LIN {X 0,Y 368.852,Z 294.537,A -85,B 0,C 180,E1 -12651.37,E2 -12651.37} C_VEL
LIN {X 0,Y 368.906,Z 294.528,A -85,B 0,C 180,E1 -12655.15,E2 -12655.15} C_VEL
LIN {X 0,Y 368.892,Z 294.531,A -85,B 0,C 180,E1 -12659.049,E2 -12659.049} C_VEL
LIN {X 0,Y 368.954,Z 294.672,A -85,B 0,C 180,E1 -12660.004,E2 -12660.004} C_VEL
LIN {X 0,Y 372.447,Z 310.54,A -85,B 0,C 180,E1 -12663.38,E2 -12663.38} C_VEL
LIN {X 0,Y 373.826,Z 317.106,A -85,B 0,C 180,E1 -12664.734,E2 -12664.734} C_VEL
LIN {X 0,Y 372.805,Z 329.127,A -85,B 0,C 180,E1 -12666.984,E2 -12666.984} C_VEL
LIN {X 0,Y 371.4,Z 344.319,A -85,B 0,C 180,E1 -12669.802,E2 -12669.802} C_VEL
LIN {X 0,Y 374.275,Z 369.679,A -85,B 0,C 180,E1 -12670.516,E2 -12670.516} C_VEL
LIN {X 0,Y 372.854,Z 448.591,A -85,B 0,C 180,E1 -12672.239,E2 -12672.239} C_VEL
LIN {X 0,Y 372.479,Z 458.52,A -85,B 0,C 180,E1 -12672.575,E2 -12672.575} C_VEL
LIN {X 0,Y 371.991,Z 468.474,A -85,B 0,C 180,E1 -12673.047,E2 -12673.047} C_VEL
LIN {X 0,Y 371.44,Z 478.285,A -85,B 0,C 180,E1 -12673.657,E2 -12673.657} C_VEL
LIN {X 0,Y 370.84,Z 487.072,A -85,B 0,C 180,E1 -12674.336,E2 -12674.336} C_VEL
LIN {X 0,Y 370.263,Z 496.307,A -85,B 0,C 180,E1 -12675.213,E2 -12675.213} C_VEL
LIN {X 0,Y 369.643,Z 505.373,A -85,B 0,C 180,E1 -12676.26,E2 -12676.26} C_VEL
LIN {X 0,Y 369.043,Z 513.274,A -85,B 0,C 180,E1 -12677.353,E2 -12677.353} C_VEL
LIN {X 0,Y 368.613,Z 520.037,A -85,B 0,C 180,E1 -12678.455,E2 -12678.455} C_VEL
LIN {X 0,Y 368.156,Z 527.063,A -85,B 0,C 180,E1 -12679.833,E2 -12679.833} C_VEL
LIN {X 0,Y 367.85,Z 532.892,A -85,B 0,C 180,E1 -12681.211,E2 -12681.211} C_VEL
LIN {X 0,Y 367.65,Z 538.484,A -85,B 0,C 180,E1 -12682.865,E2 -12682.865} C_VEL
LIN {X 0,Y 367.522,Z 542.81,A -85,B 0,C 180,E1 -12684.516,E2 -12684.516} C_VEL
LIN {X 0,Y 367.546,Z 545.139,A -85,B 0,C 180,E1 -12685.616,E2 -12685.616} C_VEL
LIN {X 0,Y 367.621,Z 548.134,A -85,B 0,C 180,E1 -12687.811,E2 -12687.811} C_VEL
LIN {X 0,Y 367.594,Z 549.066,A -85,B 0,C 180,E1 -12688.907,E2 -12688.907} C_VEL
LIN {X 0,Y 367.581,Z 549.404,A -85,B 0,C 180,E1 -12691.098,E2 -12691.098} C_VEL
LIN {X 0,Y 367.525,Z 549.003,A -85,B 0,C 180,E1 -12692.194,E2 -12692.194} C_VEL
LIN {X 0,Y 367.479,Z 546.759,A -85,B 0,C 180,E1 -12694.389,E2 -12694.389} C_VEL
LIN {X 0,Y 367.484,Z 543.958,A -85,B 0,C 180,E1 -12696.027,E2 -12696.027} C_VEL
LIN {X 0,Y 367.679,Z 540.021,A -85,B 0,C 180,E1 -12697.691,E2 -12697.691} C_VEL
LIN {X 0,Y 367.968,Z 534.919,A -85,B 0,C 180,E1 -12699.344,E2 -12699.344} C_VEL
LIN {X 0,Y 368.394,Z 529.681,A -85,B 0,C 180,E1 -12700.721,E2 -12700.721} C_VEL
LIN {X 0,Y 369.051,Z 523.384,A -85,B 0,C 180,E1 -12702.093,E2 -12702.093} C_VEL
LIN {X 0,Y 369.786,Z 515.786,A -85,B 0,C 180,E1 -12703.464,E2 -12703.464} C_VEL
LIN {X 0,Y 370.598,Z 507.776,A -85,B 0,C 180,E1 -12704.666,E2 -12704.666} C_VEL
LIN {X 0,Y 371.53,Z 498.815,A -85,B 0,C 180,E1 -12705.779,E2 -12705.779} C_VEL
LIN {X 0,Y 372.409,Z 489.59,A -85,B 0,C 180,E1 -12706.726,E2 -12706.726} C_VEL
LIN {X 0,Y 373.338,Z 479.941,A -85,B 0,C 180,E1 -12707.53,E2 -12707.53} C_VEL
LIN {X 0,Y 374.156,Z 469.906,A -85,B 0,C 180,E1 -12708.197,E2 -12708.197} C_VEL
LIN {X 0,Y 374.823,Z 459.494,A -85,B 0,C 180,E1 -12708.73,E2 -12708.73} C_VEL
LIN {X 0,Y 375.383,Z 449.742,A -85,B 0,C 180,E1 -12709.09,E2 -12709.09} C_VEL
LIN {X 0,Y 376.048,Z 423.849,A -85,B 0,C 180,E1 -12709.706,E2 -12709.706} C_VEL
LIN {X 0,Y 377.433,Z 369.357,A -85,B 0,C 180,E1 -12710.955,E2 -12710.955} C_VEL
LIN {X 0,Y 374.759,Z 350.204,A -85,B 0,C 180,E1 -12711.646,E2 -12711.646} C_VEL
LIN {X 0,Y 373.55,Z 343.29,A -85,B 0,C 180,E1 -12711.944,E2 -12711.944} C_VEL
LIN {X 0,Y 375.579,Z 321.567,A -85,B 0,C 180,E1 -12715.738,E2 -12715.738} C_VEL
LIN {X 0,Y 374.001,Z 312.86,A -85,B 0,C 180,E1 -12717.513,E2 -12717.513} C_VEL
LIN {X 0,Y 371.33,Z 302.495,A -85,B 0,C 180,E1 -12719.789,E2 -12719.789} C_VEL
LIN {X 0,Y 368.908,Z 294.535,A -85,B 0,C 180,E1 -12721.713,E2 -12721.713} C_VEL
LIN {X 0,Y 368.921,Z 294.532,A -85,B 0,C 180,E1 -12725.001,E2 -12725.001} C_VEL
LIN {X 0,Y 368.899,Z 294.537,A -85,B 0,C 180,E1 -12728.639,E2 -12728.639} C_VEL
LIN {X 0,Y 368.871,Z 294.539,A -85,B 0,C 180,E1 -12732.008,E2 -12732.008} C_VEL
LIN {X 0,Y 368.868,Z 294.539,A -85,B 0,C 180,E1 -12735.175,E2 -12735.175} C_VEL
LIN {X 0,Y 368.88,Z 294.535,A -85,B 0,C 180,E1 -12738.178,E2 -12738.178} C_VEL
LIN {X 0,Y 368.897,Z 294.533,A -85,B 0,C 180,E1 -12741.358,E2 -12741.358} C_VEL
LIN {X 0,Y 368.92,Z 294.523,A -85,B 0,C 180,E1 -12745.145,E2 -12745.145} C_VEL
LIN {X 0,Y 368.913,Z 294.522,A -85,B 0,C 180,E1 -12749.046,E2 -12749.046} C_VEL
LIN {X 0,Y 368.962,Z 294.518,A -85,B 0,C 180,E1 -12751.563,E2 -12751.563} C_VEL
LIN {X 0,Y 368.94,Z 294.527,A -85,B 0,C 180,E1 -12755.224,E2 -12755.224} C_VEL
LIN {X 0,Y 368.951,Z 294.526,A -85,B 0,C 180,E1 -12758.959,E2 -12758.959} C_VEL
LIN {X 0,Y 368.97,Z 294.525,A -85,B 0,C 180,E1 -12762.257,E2 -12762.257} C_VEL
LIN {X 0,Y 369.015,Z 294.518,A -85,B 0,C 180,E1 -12766.228,E2 -12766.228} C_VEL
LIN {X 0,Y 369.046,Z 294.519,A -85,B 0,C 180,E1 -12770.132,E2 -12770.132} C_VEL
LIN {X 0,Y 369.16,Z 294.554,A -85,B 0,C 180,E1 -12772.652,E2 -12772.652} C_VEL
LIN {X 0,Y 371.658,Z 303.249,A -85,B 0,C 180,E1 -12774.575,E2 -12774.575} C_VEL
LIN {X 0,Y 373.879,Z 311.472,A -85,B 0,C 180,E1 -12776.31,E2 -12776.31} C_VEL
LIN {X 0,Y 372.861,Z 329.538,A -85,B 0,C 180,E1 -12779.461,E2 -12779.461} C_VEL
LIN {X 0,Y 372.43,Z 338.244,A -85,B 0,C 180,E1 -12780.974,E2 -12780.974} C_VEL
LIN {X 0,Y 375.936,Z 356.545,A -85,B 0,C 180,E1 -12781.789,E2 -12781.789} C_VEL
LIN {X 0,Y 377.093,Z 364.499,A -85,B 0,C 180,E1 -12782.108,E2 -12782.108} C_VEL
LIN {X 0,Y 375.003,Z 424.893,A -85,B 0,C 180,E1 -12783.728,E2 -12783.728} C_VEL
LIN {X 0,Y 374.491,Z 435.675,A -85,B 0,C 180,E1 -12784.171,E2 -12784.171} C_VEL
LIN {X 0,Y 373.795,Z 447.132,A -85,B 0,C 180,E1 -12784.842,E2 -12784.842} C_VEL
LIN {X 0,Y 373.077,Z 457.501,A -85,B 0,C 180,E1 -12785.676,E2 -12785.676} C_VEL
LIN {X 0,Y 372.37,Z 465.772,A -85,B 0,C 180,E1 -12786.503,E2 -12786.503} C_VEL
LIN {X 0,Y 371.6,Z 473.736,A -85,B 0,C 180,E1 -12787.472,E2 -12787.472} C_VEL
LIN {X 0,Y 370.891,Z 480.383,A -85,B 0,C 180,E1 -12788.445,E2 -12788.445} C_VEL
LIN {X 0,Y 370.263,Z 486.344,A -85,B 0,C 180,E1 -12789.489,E2 -12789.489} C_VEL
LIN {X 0,Y 369.628,Z 492.019,A -85,B 0,C 180,E1 -12790.684,E2 -12790.684} C_VEL
LIN {X 0,Y 369.249,Z 495.434,A -85,B 0,C 180,E1 -12791.529,E2 -12791.529} C_VEL
LIN {X 0,Y 368.793,Z 499.293,A -85,B 0,C 180,E1 -12792.66,E2 -12792.66} C_VEL
LIN {X 0,Y 368.434,Z 502.508,A -85,B 0,C 180,E1 -12793.828,E2 -12793.828} C_VEL
LIN {X 0,Y 368.016,Z 505.852,A -85,B 0,C 180,E1 -12795.508,E2 -12795.508} C_VEL
LIN {X 0,Y 367.719,Z 507.88,A -85,B 0,C 180,E1 -12797.145,E2 -12797.145} C_VEL
LIN {X 0,Y 367.609,Z 508.44,A -85,B 0,C 180,E1 -12797.812,E2 -12797.812} C_VEL
LIN {X 0,Y 367.475,Z 508.798,A -85,B 0,C 180,E1 -12798.974,E2 -12798.974} C_VEL
LIN {X 0,Y 367.448,Z 508.486,A -85,B 0,C 180,E1 -12800.423,E2 -12800.423} C_VEL
LIN {X 0,Y 367.429,Z 507.838,A -85,B 0,C 180,E1 -12801.311,E2 -12801.311} C_VEL
LIN {X 0,Y 367.55,Z 506.489,A -85,B 0,C 180,E1 -12802.485,E2 -12802.485} C_VEL
LIN {X 0,Y 367.696,Z 504.51,A -85,B 0,C 180,E1 -12803.666,E2 -12803.666} C_VEL
LIN {X 0,Y 367.829,Z 501.801,A -85,B 0,C 180,E1 -12804.857,E2 -12804.857} C_VEL
LIN {X 0,Y 368.046,Z 497.943,A -85,B 0,C 180,E1 -12806.177,E2 -12806.177} C_VEL
LIN {X 0,Y 368.437,Z 491.446,A -85,B 0,C 180,E1 -12807.863,E2 -12807.863} C_VEL
LIN {X 0,Y 368.84,Z 485.092,A -85,B 0,C 180,E1 -12809.165,E2 -12809.165} C_VEL
LIN {X 0,Y 369.281,Z 478.413,A -85,B 0,C 180,E1 -12810.288,E2 -12810.288} C_VEL
LIN {X 0,Y 369.782,Z 470.965,A -85,B 0,C 180,E1 -12811.326,E2 -12811.326} C_VEL
LIN {X 0,Y 370.357,Z 461.379,A -85,B 0,C 180,E1 -12812.418,E2 -12812.418} C_VEL
LIN {X 0,Y 370.87,Z 450.933,A -85,B 0,C 180,E1 -12813.337,E2 -12813.337} C_VEL
LIN {X 0,Y 371.343,Z 442.01,A -85,B 0,C 180,E1 -12813.95,E2 -12813.95} C_VEL
LIN {X 0,Y 371.712,Z 431.539,A -85,B 0,C 180,E1 -12814.496,E2 -12814.496} C_VEL
LIN {X 0,Y 371.961,Z 421.603,A -85,B 0,C 180,E1 -12814.86,E2 -12814.86} C_VEL
LIN {X 0,Y 373.105,Z 361.779,A -85,B 0,C 180,E1 -12816.312,E2 -12816.312} C_VEL
LIN {X 0,Y 370.041,Z 339.575,A -85,B 0,C 180,E1 -12816.982,E2 -12816.982} C_VEL
LIN {X 0,Y 370.885,Z 325.677,A -85,B 0,C 180,E1 -12820.112,E2 -12820.112} C_VEL
LIN {X 0,Y 371.83,Z 312.012,A -85,B 0,C 180,E1 -12823.249,E2 -12823.249} C_VEL
LIN {X 0,Y 371.695,Z 308.56,A -85,B 0,C 180,E1 -12824.072,E2 -12824.072} C_VEL
LIN {X 0,Y 369.089,Z 295.334,A -85,B 0,C 180,E1 -12827.423,E2 -12827.423} C_VEL
LIN {X 0,Y 368.917,Z 294.532,A -85,B 0,C 180,E1 -12827.657,E2 -12827.657} C_VEL
LIN {X 0,Y 368.873,Z 294.538,A -85,B 0,C 180,E1 -12831.368,E2 -12831.368} C_VEL
LIN {X 0,Y 368.928,Z 294.526,A -85,B 0,C 180,E1 -12835.147,E2 -12835.147} C_VEL
LIN {X 0,Y 368.896,Z 294.529,A -85,B 0,C 180,E1 -12839.044,E2 -12839.044} C_VEL
LIN {X 0,Y 368.908,Z 294.529,A -85,B 0,C 180,E1 -12841.558,E2 -12841.558} C_VEL
LIN {X 0,Y 368.921,Z 294.531,A -85,B 0,C 180,E1 -12844.014,E2 -12844.014} C_VEL
LIN {X 0,Y 368.899,Z 294.529,A -85,B 0,C 180,E1 -12847.603,E2 -12847.603} C_VEL
LIN {X 0,Y 368.953,Z 294.524,A -85,B 0,C 180,E1 -12851.105,E2 -12851.105} C_VEL
LIN {X 0,Y 368.998,Z 294.52,A -85,B 0,C 180,E1 -12854.535,E2 -12854.535} C_VEL
LIN {X 0,Y 369.063,Z 294.513,A -85,B 0,C 180,E1 -12856.79,E2 -12856.79} C_VEL
LIN {X 0,Y 369.065,Z 294.508,A -85,B 0,C 180,E1 -12860.13,E2 -12860.13} C_VEL
LIN {X 0,Y 369.16,Z 294.503,A -85,B 0,C 180,E1 -12863.439,E2 -12863.439} C_VEL
LIN {X 0,Y 369.299,Z 294.484,A -85,B 0,C 180,E1 -12867.817,E2 -12867.817} C_VEL
LIN {X 0,Y 369.205,Z 294.491,A -85,B 0,C 180,E1 -12871.088,E2 -12871.088} C_VEL
LIN {X 0,Y 369.298,Z 294.482,A -85,B 0,C 180,E1 -12872.179,E2 -12872.179} C_VEL
LIN {X 0,Y 369.156,Z 294.499,A -85,B 0,C 180,E1 -12876.556,E2 -12876.556} C_VEL
LIN {X 0,Y 369.06,Z 294.511,A -85,B 0,C 180,E1 -12879.865,E2 -12879.865} C_VEL
LIN {X 0,Y 369.036,Z 294.512,A -85,B 0,C 180,E1 -12883.769,E2 -12883.769} C_VEL
LIN {X 0,Y 368.962,Z 294.526,A -85,B 0,C 180,E1 -12886.694,E2 -12886.694} C_VEL
LIN {X 0,Y 368.276,Z 294.607,A -85,B 0,C 180,E1 -12887.604,E2 -12887.604} C_VEL
LIN {X 0,Y 365.402,Z 294.969,A -85,B 0,C 180,E1 -12889.084,E2 -12889.084} C_VEL
LIN {X 0,Y 362.976,Z 295.272,A -85,B 0,C 180,E1 -12890.281,E2 -12890.281} C_VEL
LIN {X 0,Y 361.934,Z 295.401,A -85,B 0,C 180,E1 -12891.207,E2 -12891.207} C_VEL
LIN {X 0,Y 361.849,Z 295.408,A -85,B 0,C 180,E1 -12891.521,E2 -12891.521} C_VEL
LIN {X 0,Y 361.873,Z 295.41,A -85,B 0,C 180,E1 -12895.289,E2 -12895.289} C_VEL
LIN {X 0,Y 361.843,Z 295.411,A -85,B 0,C 180,E1 -12899.069,E2 -12899.069} C_VEL
LIN {X 0,Y 361.833,Z 295.41,A -85,B 0,C 180,E1 -12902.94,E2 -12902.94} C_VEL
LIN {X 0,Y 361.85,Z 295.412,A -85,B 0,C 180,E1 -12905.632,E2 -12905.632} C_VEL
LIN {X 0,Y 361.843,Z 295.408,A -85,B 0,C 180,E1 -12909.02,E2 -12909.02} C_VEL
LIN {X 0,Y 361.809,Z 295.413,A -85,B 0,C 180,E1 -12912.824,E2 -12912.824} C_VEL
LIN {X 0,Y 361.79,Z 295.417,A -85,B 0,C 180,E1 -12915.942,E2 -12915.942} C_VEL
LIN {X 0,Y 361.804,Z 295.413,A -85,B 0,C 180,E1 -12919.24,E2 -12919.24} C_VEL
LIN {X 0,Y 361.827,Z 295.417,A -85,B 0,C 180,E1 -12922.773,E2 -12922.773} C_VEL
LIN {X 0,Y 361.814,Z 295.412,A -85,B 0,C 180,E1 -12925.715,E2 -12925.715} C_VEL
LIN {X 0,Y 361.837,Z 295.41,A -85,B 0,C 180,E1 -12929.668,E2 -12929.668} C_VEL
LIN {X 0,Y 361.913,Z 295.405,A -85,B 0,C 180,E1 -12933.471,E2 -12933.471} C_VEL
LIN {X 0,Y 361.834,Z 295.411,A -85,B 0,C 180,E1 -12937.14,E2 -12937.14} C_VEL
LIN {X 0,Y 361.82,Z 295.41,A -85,B 0,C 180,E1 -12940.718,E2 -12940.718} C_VEL
LIN {X 0,Y 361.895,Z 295.406,A -85,B 0,C 180,E1 -12944.223,E2 -12944.223} C_VEL
LIN {X 0,Y 361.951,Z 295.397,A -85,B 0,C 180,E1 -12946.525,E2 -12946.525} C_VEL
LIN {X 0,Y 361.984,Z 295.393,A -85,B 0,C 180,E1 -12949.936,E2 -12949.936} C_VEL
LIN {X 0,Y 362.112,Z 295.374,A -85,B 0,C 180,E1 -12953.312,E2 -12953.312} C_VEL
LIN {X 0,Y 362.236,Z 295.359,A -85,B 0,C 180,E1 -12957.776,E2 -12957.776} C_VEL
LIN {X 0,Y 362.374,Z 295.342,A -85,B 0,C 180,E1 -12959.999,E2 -12959.999} C_VEL
LIN {X 0,Y 362.23,Z 295.36,A -85,B 0,C 180,E1 -12962.223,E2 -12962.223} C_VEL
LIN {X 0,Y 362.111,Z 295.376,A -85,B 0,C 180,E1 -12966.687,E2 -12966.687} C_VEL
LIN {X 0,Y 361.981,Z 295.392,A -85,B 0,C 180,E1 -12970.063,E2 -12970.063} C_VEL
LIN {X 0,Y 361.949,Z 295.399,A -85,B 0,C 180,E1 -12973.899,E2 -12973.899} C_VEL
LIN {X 0,Y 361.92,Z 295.405,A -85,B 0,C 180,E1 -12977.94,E2 -12977.94} C_VEL
LIN {X 0,Y 361.837,Z 295.41,A -85,B 0,C 180,E1 -12981.656,E2 -12981.656} C_VEL
LIN {X 0,Y 361.882,Z 295.403,A -85,B 0,C 180,E1 -12985.293,E2 -12985.293} C_VEL
LIN {X 0,Y 361.862,Z 295.406,A -85,B 0,C 180,E1 -12987.782,E2 -12987.782} C_VEL
LIN {X 0,Y 361.792,Z 295.414,A -85,B 0,C 180,E1 -12991.633,E2 -12991.633} C_VEL
LIN {X 0,Y 361.835,Z 295.411,A -85,B 0,C 180,E1 -12995.348,E2 -12995.348} C_VEL
LIN {X 0,Y 361.827,Z 295.416,A -85,B 0,C 180,E1 -12999.029,E2 -12999.029} C_VEL
LIN {X 0,Y 361.802,Z 295.415,A -85,B 0,C 180,E1 -13002.833,E2 -13002.833} C_VEL
LIN {X 0,Y 361.785,Z 295.417,A -85,B 0,C 180,E1 -13005.951,E2 -13005.951} C_VEL
LIN {X 0,Y 361.805,Z 295.415,A -85,B 0,C 180,E1 -13009.249,E2 -13009.249} C_VEL
LIN {X 0,Y 361.835,Z 295.409,A -85,B 0,C 180,E1 -13012.985,E2 -13012.985} C_VEL
LIN {X 0,Y 361.835,Z 295.411,A -85,B 0,C 180,E1 -13016.635,E2 -13016.635} C_VEL
LIN {X 0,Y 361.89,Z 295.489,A -85,B 0,C 180,E1 -13019.679,E2 -13019.679} C_VEL
LIN {X 0,Y 365.13,Z 310.229,A -85,B 0,C 180,E1 -13022.886,E2 -13022.886} C_VEL
LIN {X 0,Y 366.901,Z 318.921,A -85,B 0,C 180,E1 -13024.712,E2 -13024.712} C_VEL
LIN {X 0,Y 365.132,Z 337.578,A -85,B 0,C 180,E1 -13028.257,E2 -13028.257} C_VEL
LIN {X 0,Y 364.455,Z 344.417,A -85,B 0,C 180,E1 -13029.547,E2 -13029.547} C_VEL
LIN {X 0,Y 367.345,Z 370.807,A -85,B 0,C 180,E1 -13030.286,E2 -13030.286} C_VEL
LIN {X 0,Y 365.895,Z 448.793,A -85,B 0,C 180,E1 -13032.034,E2 -13032.034} C_VEL
LIN {X 0,Y 365.517,Z 458.547,A -85,B 0,C 180,E1 -13032.376,E2 -13032.376} C_VEL
LIN {X 0,Y 365.015,Z 468.409,A -85,B 0,C 180,E1 -13032.857,E2 -13032.857} C_VEL
LIN {X 0,Y 364.448,Z 478.164,A -85,B 0,C 180,E1 -13033.479,E2 -13033.479} C_VEL
LIN {X 0,Y 363.837,Z 486.913,A -85,B 0,C 180,E1 -13034.17,E2 -13034.17} C_VEL
LIN {X 0,Y 363.201,Z 496.869,A -85,B 0,C 180,E1 -13035.148,E2 -13035.148} C_VEL
LIN {X 0,Y 362.628,Z 504.665,A -85,B 0,C 180,E1 -13036.064,E2 -13036.064} C_VEL
LIN {X 0,Y 362.044,Z 512.174,A -85,B 0,C 180,E1 -13037.104,E2 -13037.104} C_VEL
LIN {X 0,Y 361.48,Z 520.509,A -85,B 0,C 180,E1 -13038.508,E2 -13038.508} C_VEL
LIN {X 0,Y 361.043,Z 527.396,A -85,B 0,C 180,E1 -13039.913,E2 -13039.913} C_VEL
LIN {X 0,Y 360.783,Z 532.112,A -85,B 0,C 180,E1 -13041.038,E2 -13041.038} C_VEL
LIN {X 0,Y 360.577,Z 537.794,A -85,B 0,C 180,E1 -13042.725,E2 -13042.725} C_VEL
LIN {X 0,Y 360.438,Z 542.193,A -85,B 0,C 180,E1 -13044.408,E2 -13044.408} C_VEL
LIN {X 0,Y 360.48,Z 544.54,A -85,B 0,C 180,E1 -13045.53,E2 -13045.53} C_VEL
LIN {X 0,Y 360.537,Z 547.644,A -85,B 0,C 180,E1 -13047.768,E2 -13047.768} C_VEL
LIN {X 0,Y 360.529,Z 548.586,A -85,B 0,C 180,E1 -13048.885,E2 -13048.885} C_VEL
LIN {X 0,Y 360.515,Z 549.019,A -85,B 0,C 180,E1 -13051.119,E2 -13051.119} C_VEL
LIN {X 0,Y 360.427,Z 548.613,A -85,B 0,C 180,E1 -13052.237,E2 -13052.237} C_VEL
LIN {X 0,Y 360.386,Z 546.46,A -85,B 0,C 180,E1 -13054.476,E2 -13054.476} C_VEL
LIN {X 0,Y 360.382,Z 544.064,A -85,B 0,C 180,E1 -13055.975,E2 -13055.975} C_VEL
LIN {X 0,Y 360.607,Z 539.811,A -85,B 0,C 180,E1 -13057.843,E2 -13057.843} C_VEL
LIN {X 0,Y 360.931,Z 534.778,A -85,B 0,C 180,E1 -13059.528,E2 -13059.528} C_VEL
LIN {X 0,Y 361.388,Z 529.619,A -85,B 0,C 180,E1 -13060.931,E2 -13060.931} C_VEL
LIN {X 0,Y 362.098,Z 523.387,A -85,B 0,C 180,E1 -13062.329,E2 -13062.329} C_VEL
LIN {X 0,Y 362.863,Z 515.856,A -85,B 0,C 180,E1 -13063.726,E2 -13063.726} C_VEL
LIN {X 0,Y 363.711,Z 507.909,A -85,B 0,C 180,E1 -13064.952,E2 -13064.952} C_VEL
LIN {X 0,Y 364.717,Z 499.054,A -85,B 0,C 180,E1 -13066.082,E2 -13066.082} C_VEL
LIN {X 0,Y 365.651,Z 489.947,A -85,B 0,C 180,E1 -13067.045,E2 -13067.045} C_VEL
LIN {X 0,Y 366.618,Z 480.522,A -85,B 0,C 180,E1 -13067.862,E2 -13067.862} C_VEL
LIN {X 0,Y 367.561,Z 469.647,A -85,B 0,C 180,E1 -13068.607,E2 -13068.607} C_VEL
LIN {X 0,Y 368.26,Z 459.364,A -85,B 0,C 180,E1 -13069.148,E2 -13069.148} C_VEL
LIN {X 0,Y 368.867,Z 448.662,A -85,B 0,C 180,E1 -13069.55,E2 -13069.55} C_VEL
LIN {X 0,Y 369.763,Z 418.32,A -85,B 0,C 180,E1 -13070.272,E2 -13070.272} C_VEL
LIN {X 0,Y 371.004,Z 369.957,A -85,B 0,C 180,E1 -13071.415,E2 -13071.415} C_VEL
LIN {X 0,Y 368.495,Z 351.79,A -85,B 0,C 180,E1 -13072.101,E2 -13072.101} C_VEL
LIN {X 0,Y 366.974,Z 343.172,A -85,B 0,C 180,E1 -13072.489,E2 -13072.489} C_VEL
LIN {X 0,Y 368.932,Z 323.532,A -85,B 0,C 180,E1 -13075.985,E2 -13075.985} C_VEL
LIN {X 0,Y 367.259,Z 314.592,A -85,B 0,C 180,E1 -13077.873,E2 -13077.873} C_VEL
LIN {X 0,Y 364.349,Z 303.535,A -85,B 0,C 180,E1 -13080.405,E2 -13080.405} C_VEL
LIN {X 0,Y 361.852,Z 295.413,A -85,B 0,C 180,E1 -13082.447,E2 -13082.447} C_VEL
LIN {X 0,Y 361.86,Z 295.413,A -85,B 0,C 180,E1 -13085.636,E2 -13085.636} C_VEL
LIN {X 0,Y 361.86,Z 295.415,A -85,B 0,C 180,E1 -13089.026,E2 -13089.026} C_VEL
LIN {X 0,Y 361.826,Z 295.417,A -85,B 0,C 180,E1 -13092.828,E2 -13092.828} C_VEL
LIN {X 0,Y 361.806,Z 295.416,A -85,B 0,C 180,E1 -13095.946,E2 -13095.946} C_VEL
LIN {X 0,Y 361.856,Z 295.411,A -85,B 0,C 180,E1 -13099.238,E2 -13099.238} C_VEL
LIN {X 0,Y 361.853,Z 295.406,A -85,B 0,C 180,E1 -13102.981,E2 -13102.981} C_VEL
LIN {X 0,Y 361.842,Z 295.403,A -85,B 0,C 180,E1 -13106.63,E2 -13106.63} C_VEL
LIN {X 0,Y 361.858,Z 295.4,A -85,B 0,C 180,E1 -13109.671,E2 -13109.671} C_VEL
LIN {X 0,Y 361.935,Z 295.397,A -85,B 0,C 180,E1 -13113.474,E2 -13113.474} C_VEL
LIN {X 0,Y 361.888,Z 295.408,A -85,B 0,C 180,E1 -13117.145,E2 -13117.145} C_VEL
LIN {X 0,Y 361.911,Z 295.403,A -85,B 0,C 180,E1 -13120.724,E2 -13120.724} C_VEL
LIN {X 0,Y 361.923,Z 295.402,A -85,B 0,C 180,E1 -13124.226,E2 -13124.226} C_VEL
LIN {X 0,Y 361.977,Z 295.396,A -85,B 0,C 180,E1 -13126.528,E2 -13126.528} C_VEL
LIN {X 0,Y 362.01,Z 295.396,A -85,B 0,C 180,E1 -13129.938,E2 -13129.938} C_VEL
LIN {X 0,Y 362.135,Z 295.534,A -85,B 0,C 180,E1 -13131.954,E2 -13131.954} C_VEL
LIN {X 0,Y 365.035,Z 305.197,A -85,B 0,C 180,E1 -13134.199,E2 -13134.199} C_VEL
LIN {X 0,Y 367.348,Z 314.468,A -85,B 0,C 180,E1 -13136.2,E2 -13136.2} C_VEL
LIN {X 0,Y 366.089,Z 334.351,A -85,B 0,C 180,E1 -13139.726,E2 -13139.726} C_VEL
LIN {X 0,Y 365.832,Z 338.257,A -85,B 0,C 180,E1 -13140.413,E2 -13140.413} C_VEL
LIN {X 0,Y 369.455,Z 356.953,A -85,B 0,C 180,E1 -13141.304,E2 -13141.304} C_VEL
LIN {X 0,Y 370.657,Z 365.769,A -85,B 0,C 180,E1 -13141.663,E2 -13141.663} C_VEL
LIN {X 0,Y 368.478,Z 425.757,A -85,B 0,C 180,E1 -13143.315,E2 -13143.315} C_VEL
LIN {X 0,Y 367.891,Z 437.742,A -85,B 0,C 180,E1 -13143.834,E2 -13143.834} C_VEL
LIN {X 0,Y 367.057,Z 449.679,A -85,B 0,C 180,E1 -13144.608,E2 -13144.608} C_VEL
LIN {X 0,Y 366.383,Z 458.543,A -85,B 0,C 180,E1 -13145.356,E2 -13145.356} C_VEL
LIN {X 0,Y 365.615,Z 466.762,A -85,B 0,C 180,E1 -13146.208,E2 -13146.208} C_VEL
LIN {X 0,Y 364.783,Z 474.609,A -85,B 0,C 180,E1 -13147.195,E2 -13147.195} C_VEL
LIN {X 0,Y 363.949,Z 482.061,A -85,B 0,C 180,E1 -13148.328,E2 -13148.328} C_VEL
LIN {X 0,Y 363.068,Z 489.887,A -85,B 0,C 180,E1 -13149.805,E2 -13149.805} C_VEL
LIN {X 0,Y 362.375,Z 495.583,A -85,B 0,C 180,E1 -13151.184,E2 -13151.184} C_VEL
LIN {X 0,Y 361.858,Z 499.502,A -85,B 0,C 180,E1 -13152.336,E2 -13152.336} C_VEL
LIN {X 0,Y 361.343,Z 503.801,A -85,B 0,C 180,E1 -13154.014,E2 -13154.014} C_VEL
LIN {X 0,Y 360.868,Z 506.998,A -85,B 0,C 180,E1 -13155.823,E2 -13155.823} C_VEL
LIN {X 0,Y 360.613,Z 508.531,A -85,B 0,C 180,E1 -13157.272,E2 -13157.272} C_VEL
LIN {X 0,Y 360.475,Z 509.069,A -85,B 0,C 180,E1 -13158.177,E2 -13158.177} C_VEL
LIN {X 0,Y 360.377,Z 509.271,A -85,B 0,C 180,E1 -13159.362,E2 -13159.362} C_VEL
LIN {X 0,Y 360.357,Z 508.799,A -85,B 0,C 180,E1 -13160.596,E2 -13160.596} C_VEL
LIN {X 0,Y 360.388,Z 507.747,A -85,B 0,C 180,E1 -13161.748,E2 -13161.748} C_VEL
LIN {X 0,Y 360.598,Z 504.893,A -85,B 0,C 180,E1 -13163.656,E2 -13163.656} C_VEL
LIN {X 0,Y 360.806,Z 500.774,A -85,B 0,C 180,E1 -13165.375,E2 -13165.375} C_VEL
LIN {X 0,Y 361.123,Z 495.855,A -85,B 0,C 180,E1 -13166.904,E2 -13166.904} C_VEL
LIN {X 0,Y 361.414,Z 490.886,A -85,B 0,C 180,E1 -13168.136,E2 -13168.136} C_VEL
LIN {X 0,Y 361.814,Z 484.819,A -85,B 0,C 180,E1 -13169.372,E2 -13169.372} C_VEL
LIN {X 0,Y 362.406,Z 476.428,A -85,B 0,C 180,E1 -13170.763,E2 -13170.763} C_VEL
LIN {X 0,Y 363.011,Z 466.833,A -85,B 0,C 180,E1 -13172.005,E2 -13172.005} C_VEL
LIN {X 0,Y 363.587,Z 457.853,A -85,B 0,C 180,E1 -13172.933,E2 -13172.933} C_VEL
LIN {X 0,Y 364.052,Z 448.472,A -85,B 0,C 180,E1 -13173.713,E2 -13173.713} C_VEL
LIN {X 0,Y 364.484,Z 438.919,A -85,B 0,C 180,E1 -13174.334,E2 -13174.334} C_VEL
LIN {X 0,Y 364.902,Z 426.577,A -85,B 0,C 180,E1 -13174.917,E2 -13174.917} C_VEL
LIN {X 0,Y 365.329,Z 408.302,A -85,B 0,C 180,E1 -13175.413,E2 -13175.413} C_VEL
LIN {X 0,Y 366.145,Z 362.498,A -85,B 0,C 180,E1 -13176.544,E2 -13176.544} C_VEL
LIN {X 0,Y 363.116,Z 339.521,A -85,B 0,C 180,E1 -13177.274,E2 -13177.274} C_VEL
LIN {X 0,Y 364.293,Z 321.474,A -85,B 0,C 180,E1 -13181.422,E2 -13181.422} C_VEL
LIN {X 0,Y 364.866,Z 310.928,A -85,B 0,C 180,E1 -13183.903,E2 -13183.903} C_VEL
LIN {X 0,Y 362.627,Z 299.172,A -85,B 0,C 180,E1 -13186.91,E2 -13186.91} C_VEL
LIN {X 0,Y 361.855,Z 295.41,A -85,B 0,C 180,E1 -13187.916,E2 -13187.916} C_VEL
LIN {X 0,Y 361.839,Z 295.415,A -85,B 0,C 180,E1 -13191.573,E2 -13191.573} C_VEL
LIN {X 0,Y 361.868,Z 295.405,A -85,B 0,C 180,E1 -13194.658,E2 -13194.658} C_VEL
LIN {X 0,Y 361.834,Z 295.411,A -85,B 0,C 180,E1 -13198.371,E2 -13198.371} C_VEL
LIN {X 0,Y 361.85,Z 295.407,A -85,B 0,C 180,E1 -13200.951,E2 -13200.951} C_VEL
LIN {X 0,Y 361.854,Z 295.409,A -85,B 0,C 180,E1 -13204.705,E2 -13204.705} C_VEL
LIN {X 0,Y 361.857,Z 295.412,A -85,B 0,C 180,E1 -13208.345,E2 -13208.345} C_VEL
LIN {X 0,Y 361.924,Z 295.399,A -85,B 0,C 180,E1 -13212.085,E2 -13212.085} C_VEL
LIN {X 0,Y 362.004,Z 295.388,A -85,B 0,C 180,E1 -13216.101,E2 -13216.101} C_VEL
LIN {X 0,Y 362.002,Z 295.388,A -85,B 0,C 180,E1 -13219.936,E2 -13219.936} C_VEL
LIN {X 0,Y 362.124,Z 295.38,A -85,B 0,C 180,E1 -13223.311,E2 -13223.311} C_VEL
LIN {X 0,Y 362.261,Z 295.361,A -85,B 0,C 180,E1 -13227.774,E2 -13227.774} C_VEL
LIN {X 0,Y 362.177,Z 295.367,A -85,B 0,C 180,E1 -13231.11,E2 -13231.11} C_VEL
LIN {X 0,Y 362.261,Z 295.359,A -85,B 0,C 180,E1 -13232.221,E2 -13232.221} C_VEL
LIN {X 0,Y 362.12,Z 295.375,A -85,B 0,C 180,E1 -13236.684,E2 -13236.684} C_VEL
LIN {X 0,Y 361.997,Z 295.393,A -85,B 0,C 180,E1 -13240.06,E2 -13240.06} C_VEL
LIN {X 0,Y 361.997,Z 295.389,A -85,B 0,C 180,E1 -13243.895,E2 -13243.895} C_VEL
LIN {X 0,Y 361.925,Z 295.402,A -85,B 0,C 180,E1 -13246.93,E2 -13246.93} C_VEL
LIN {X 0,Y 361.881,Z 295.405,A -85,B 0,C 180,E1 -13250.457,E2 -13250.457} C_VEL
LIN {X 0,Y 361.849,Z 295.408,A -85,B 0,C 180,E1 -13251.521,E2 -13251.521} C_VEL
LIN {X 0,Y 361.177,Z 295.494,A -85,B 0,C 180,E1 -13252.451,E2 -13252.451} C_VEL
LIN {X 0,Y 358.316,Z 295.847,A -85,B 0,C 180,E1 -13253.962,E2 -13253.962} C_VEL
LIN {X 0,Y 355.897,Z 296.156,A -85,B 0,C 180,E1 -13255.185,E2 -13255.185} C_VEL
LIN {X 0,Y 354.864,Z 296.278,A -85,B 0,C 180,E1 -13256.131,E2 -13256.131} C_VEL
LIN {X 0,Y 354.783,Z 296.287,A -85,B 0,C 180,E1 -13256.452,E2 -13256.452} C_VEL
LIN {X 0,Y 354.784,Z 296.291,A -85,B 0,C 180,E1 -13259.679,E2 -13259.679} C_VEL
LIN {X 0,Y 354.772,Z 296.289,A -85,B 0,C 180,E1 -13262.329,E2 -13262.329} C_VEL
LIN {X 0,Y 354.804,Z 296.291,A -85,B 0,C 180,E1 -13265.694,E2 -13265.694} C_VEL
LIN {X 0,Y 354.804,Z 296.286,A -85,B 0,C 180,E1 -13269.419,E2 -13269.419} C_VEL
LIN {X 0,Y 354.762,Z 296.291,A -85,B 0,C 180,E1 -13272.862,E2 -13272.862} C_VEL
LIN {X 0,Y 354.739,Z 296.297,A -85,B 0,C 180,E1 -13276.098,E2 -13276.098} C_VEL
LIN {X 0,Y 354.757,Z 296.292,A -85,B 0,C 180,E1 -13279.174,E2 -13279.174} C_VEL
LIN {X 0,Y 354.773,Z 296.292,A -85,B 0,C 180,E1 -13282.399,E2 -13282.399} C_VEL
LIN {X 0,Y 354.773,Z 296.295,A -85,B 0,C 180,E1 -13284.936,E2 -13284.936} C_VEL
LIN {X 0,Y 354.755,Z 296.291,A -85,B 0,C 180,E1 -13288.401,E2 -13288.401} C_VEL
LIN {X 0,Y 354.812,Z 296.287,A -85,B 0,C 180,E1 -13291.615,E2 -13291.615} C_VEL
LIN {X 0,Y 354.856,Z 296.278,A -85,B 0,C 180,E1 -13294.169,E2 -13294.169} C_VEL
LIN {X 0,Y 354.771,Z 296.293,A -85,B 0,C 180,E1 -13297.889,E2 -13297.889} C_VEL
LIN {X 0,Y 354.818,Z 296.289,A -85,B 0,C 180,E1 -13301.919,E2 -13301.919} C_VEL
LIN {X 0,Y 354.871,Z 296.276,A -85,B 0,C 180,E1 -13305.08,E2 -13305.08} C_VEL
LIN {X 0,Y 354.889,Z 296.277,A -85,B 0,C 180,E1 -13308.577,E2 -13308.577} C_VEL
LIN {X 0,Y 355.033,Z 296.259,A -85,B 0,C 180,E1 -13312.034,E2 -13312.034} C_VEL
LIN {X 0,Y 355.039,Z 296.26,A -85,B 0,C 180,E1 -13314.319,E2 -13314.319} C_VEL
LIN {X 0,Y 355.2,Z 296.235,A -85,B 0,C 180,E1 -13317.731,E2 -13317.731} C_VEL
LIN {X 0,Y 355.323,Z 296.22,A -85,B 0,C 180,E1 -13319.999,E2 -13319.999} C_VEL
LIN {X 0,Y 355.194,Z 296.236,A -85,B 0,C 180,E1 -13322.267,E2 -13322.267} C_VEL
LIN {X 0,Y 355.074,Z 296.253,A -85,B 0,C 180,E1 -13326.82,E2 -13326.82} C_VEL
LIN {X 0,Y 354.928,Z 296.269,A -85,B 0,C 180,E1 -13330.265,E2 -13330.265} C_VEL
LIN {X 0,Y 354.893,Z 296.277,A -85,B 0,C 180,E1 -13334.019,E2 -13334.019} C_VEL
LIN {X 0,Y 354.875,Z 296.281,A -85,B 0,C 180,E1 -13338.11,E2 -13338.11} C_VEL
LIN {X 0,Y 354.784,Z 296.294,A -85,B 0,C 180,E1 -13342.109,E2 -13342.109} C_VEL
LIN {X 0,Y 354.853,Z 296.28,A -85,B 0,C 180,E1 -13345.83,E2 -13345.83} C_VEL
LIN {X 0,Y 354.76,Z 296.29,A -85,B 0,C 180,E1 -13349.687,E2 -13349.687} C_VEL
LIN {X 0,Y 354.776,Z 296.288,A -85,B 0,C 180,E1 -13353.687,E2 -13353.687} C_VEL
LIN {X 0,Y 354.758,Z 296.292,A -85,B 0,C 180,E1 -13356.464,E2 -13356.464} C_VEL
LIN {X 0,Y 354.79,Z 296.29,A -85,B 0,C 180,E1 -13359.427,E2 -13359.427} C_VEL
LIN {X 0,Y 354.754,Z 296.293,A -85,B 0,C 180,E1 -13362.871,E2 -13362.871} C_VEL
LIN {X 0,Y 354.735,Z 296.295,A -85,B 0,C 180,E1 -13366.107,E2 -13366.107} C_VEL
LIN {X 0,Y 354.757,Z 296.292,A -85,B 0,C 180,E1 -13369.183,E2 -13369.183} C_VEL
LIN {X 0,Y 354.773,Z 296.29,A -85,B 0,C 180,E1 -13372.409,E2 -13372.409} C_VEL
LIN {X 0,Y 354.783,Z 296.287,A -85,B 0,C 180,E1 -13374.944,E2 -13374.944} C_VEL
LIN {X 0,Y 354.772,Z 296.294,A -85,B 0,C 180,E1 -13378.41,E2 -13378.41} C_VEL
LIN {X 0,Y 354.835,Z 296.288,A -85,B 0,C 180,E1 -13379.342,E2 -13379.342} C_VEL
LIN {X 0,Y 358.089,Z 311.058,A -85,B 0,C 180,E1 -13382.625,E2 -13382.625} C_VEL
LIN {X 0,Y 359.912,Z 320.101,A -85,B 0,C 180,E1 -13384.563,E2 -13384.563} C_VEL
LIN {X 0,Y 358.302,Z 336.999,A -85,B 0,C 180,E1 -13387.848,E2 -13387.848} C_VEL
LIN {X 0,Y 357.548,Z 344.273,A -85,B 0,C 180,E1 -13389.246,E2 -13389.246} C_VEL
LIN {X 0,Y 360.444,Z 371.505,A -85,B 0,C 180,E1 -13390.043,E2 -13390.043} C_VEL
LIN {X 0,Y 358.964,Z 447.736,A -85,B 0,C 180,E1 -13391.786,E2 -13391.786} C_VEL
LIN {X 0,Y 358.608,Z 457.761,A -85,B 0,C 180,E1 -13392.136,E2 -13392.136} C_VEL
LIN {X 0,Y 358.092,Z 467.14,A -85,B 0,C 180,E1 -13392.589,E2 -13392.589} C_VEL
LIN {X 0,Y 357.557,Z 476.166,A -85,B 0,C 180,E1 -13393.151,E2 -13393.151} C_VEL
LIN {X 0,Y 356.838,Z 486.755,A -85,B 0,C 180,E1 -13393.998,E2 -13393.998} C_VEL
LIN {X 0,Y 356.173,Z 496.68,A -85,B 0,C 180,E1 -13394.994,E2 -13394.994} C_VEL
LIN {X 0,Y 355.596,Z 503.985,A -85,B 0,C 180,E1 -13395.863,E2 -13395.863} C_VEL
LIN {X 0,Y 354.916,Z 512.809,A -85,B 0,C 180,E1 -13397.132,E2 -13397.132} C_VEL
LIN {X 0,Y 354.486,Z 519.539,A -85,B 0,C 180,E1 -13398.279,E2 -13398.279} C_VEL
LIN {X 0,Y 353.979,Z 526.527,A -85,B 0,C 180,E1 -13399.71,E2 -13399.71} C_VEL
LIN {X 0,Y 353.678,Z 532.323,A -85,B 0,C 180,E1 -13401.144,E2 -13401.144} C_VEL
LIN {X 0,Y 353.497,Z 537.102,A -85,B 0,C 180,E1 -13402.578,E2 -13402.578} C_VEL
LIN {X 0,Y 353.351,Z 541.576,A -85,B 0,C 180,E1 -13404.296,E2 -13404.296} C_VEL
LIN {X 0,Y 353.412,Z 543.926,A -85,B 0,C 180,E1 -13405.44,E2 -13405.44} C_VEL
LIN {X 0,Y 353.439,Z 547.152,A -85,B 0,C 180,E1 -13407.723,E2 -13407.723} C_VEL
LIN {X 0,Y 353.466,Z 548.096,A -85,B 0,C 180,E1 -13408.863,E2 -13408.863} C_VEL
LIN {X 0,Y 353.431,Z 548.633,A -85,B 0,C 180,E1 -13411.142,E2 -13411.142} C_VEL
LIN {X 0,Y 353.329,Z 548.224,A -85,B 0,C 180,E1 -13412.282,E2 -13412.282} C_VEL
LIN {X 0,Y 353.297,Z 546.175,A -85,B 0,C 180,E1 -13414.566,E2 -13414.566} C_VEL
LIN {X 0,Y 353.311,Z 544.037,A -85,B 0,C 180,E1 -13415.967,E2 -13415.967} C_VEL
LIN {X 0,Y 353.534,Z 539.645,A -85,B 0,C 180,E1 -13418,E2 -13418} C_VEL
LIN {X 0,Y 353.909,Z 534.665,A -85,B 0,C 180,E1 -13419.719,E2 -13419.719} C_VEL
LIN {X 0,Y 354.497,Z 528.357,A -85,B 0,C 180,E1 -13421.436,E2 -13421.436} C_VEL
LIN {X 0,Y 355.284,Z 521.938,A -85,B 0,C 180,E1 -13422.859,E2 -13422.859} C_VEL
LIN {X 0,Y 355.944,Z 515.925,A -85,B 0,C 180,E1 -13423.998,E2 -13423.998} C_VEL
LIN {X 0,Y 356.979,Z 506.895,A -85,B 0,C 180,E1 -13425.414,E2 -13425.414} C_VEL
LIN {X 0,Y 358.056,Z 498.185,A -85,B 0,C 180,E1 -13426.536,E2 -13426.536} C_VEL
LIN {X 0,Y 359.087,Z 489.026,A -85,B 0,C 180,E1 -13427.513,E2 -13427.513} C_VEL
LIN {X 0,Y 360.112,Z 479.469,A -85,B 0,C 180,E1 -13428.343,E2 -13428.343} C_VEL
LIN {X 0,Y 360.988,Z 469.574,A -85,B 0,C 180,E1 -13429.033,E2 -13429.033} C_VEL
LIN {X 0,Y 361.718,Z 459.385,A -85,B 0,C 180,E1 -13429.583,E2 -13429.583} C_VEL
LIN {X 0,Y 362.366,Z 448.866,A -85,B 0,C 180,E1 -13429.989,E2 -13429.989} C_VEL
LIN {X 0,Y 363.112,Z 424.583,A -85,B 0,C 180,E1 -13430.594,E2 -13430.594} C_VEL
LIN {X 0,Y 364.639,Z 370.858,A -85,B 0,C 180,E1 -13431.898,E2 -13431.898} C_VEL
LIN {X 0,Y 362.288,Z 353.321,A -85,B 0,C 180,E1 -13432.583,E2 -13432.583} C_VEL
LIN {X 0,Y 360.442,Z 343.247,A -85,B 0,C 180,E1 -13433.031,E2 -13433.031} C_VEL
LIN {X 0,Y 362.306,Z 325.911,A -85,B 0,C 180,E1 -13436.187,E2 -13436.187} C_VEL
LIN {X 0,Y 360.973,Z 318.061,A -85,B 0,C 180,E1 -13437.857,E2 -13437.857} C_VEL
LIN {X 0,Y 358.29,Z 307.443,A -85,B 0,C 180,E1 -13440.337,E2 -13440.337} C_VEL
LIN {X 0,Y 354.801,Z 296.292,A -85,B 0,C 180,E1 -13443.217,E2 -13443.217} C_VEL
LIN {X 0,Y 354.789,Z 296.292,A -85,B 0,C 180,E1 -13446.459,E2 -13446.459} C_VEL
LIN {X 0,Y 354.816,Z 296.292,A -85,B 0,C 180,E1 -13449.423,E2 -13449.423} C_VEL
LIN {X 0,Y 354.778,Z 296.295,A -85,B 0,C 180,E1 -13452.866,E2 -13452.866} C_VEL
LIN {X 0,Y 354.755,Z 296.295,A -85,B 0,C 180,E1 -13456.103,E2 -13456.103} C_VEL
LIN {X 0,Y 354.807,Z 296.289,A -85,B 0,C 180,E1 -13459.182,E2 -13459.182} C_VEL
LIN {X 0,Y 354.794,Z 296.285,A -85,B 0,C 180,E1 -13462.402,E2 -13462.402} C_VEL
LIN {X 0,Y 354.796,Z 296.281,A -85,B 0,C 180,E1 -13464.94,E2 -13464.94} C_VEL
LIN {X 0,Y 354.777,Z 296.288,A -85,B 0,C 180,E1 -13468.405,E2 -13468.405} C_VEL
LIN {X 0,Y 354.833,Z 296.278,A -85,B 0,C 180,E1 -13471.618,E2 -13471.618} C_VEL
LIN {X 0,Y 354.88,Z 296.274,A -85,B 0,C 180,E1 -13474.172,E2 -13474.172} C_VEL
LIN {X 0,Y 354.833,Z 296.287,A -85,B 0,C 180,E1 -13477.895,E2 -13477.895} C_VEL
LIN {X 0,Y 354.903,Z 296.278,A -85,B 0,C 180,E1 -13481.891,E2 -13481.891} C_VEL
LIN {X 0,Y 354.921,Z 296.273,A -85,B 0,C 180,E1 -13485.982,E2 -13485.982} C_VEL
LIN {X 0,Y 354.958,Z 296.275,A -85,B 0,C 180,E1 -13489.736,E2 -13489.736} C_VEL
LIN {X 0,Y 355.039,Z 296.416,A -85,B 0,C 180,E1 -13491.164,E2 -13491.164} C_VEL
LIN {X 0,Y 358.162,Z 305.951,A -85,B 0,C 180,E1 -13493.522,E2 -13493.522} C_VEL
LIN {X 0,Y 360.678,Z 316.034,A -85,B 0,C 180,E1 -13495.778,E2 -13495.778} C_VEL
LIN {X 0,Y 360.675,Z 319.244,A -85,B 0,C 180,E1 -13496.389,E2 -13496.389} C_VEL
LIN {X 0,Y 359.323,Z 338.609,A -85,B 0,C 180,E1 -13499.849,E2 -13499.849} C_VEL
LIN {X 0,Y 362.907,Z 356.472,A -85,B 0,C 180,E1 -13500.737,E2 -13500.737} C_VEL
LIN {X 0,Y 364.344,Z 366.21,A -85,B 0,C 180,E1 -13501.168,E2 -13501.168} C_VEL
LIN {X 0,Y 361.95,Z 426.632,A -85,B 0,C 180,E1 -13502.887,E2 -13502.887} C_VEL
LIN {X 0,Y 361.234,Z 439.61,A -85,B 0,C 180,E1 -13503.486,E2 -13503.486} C_VEL
LIN {X 0,Y 360.48,Z 450.118,A -85,B 0,C 180,E1 -13504.193,E2 -13504.193} C_VEL
LIN {X 0,Y 359.749,Z 458.946,A -85,B 0,C 180,E1 -13504.951,E2 -13504.951} C_VEL
LIN {X 0,Y 359.005,Z 466.648,A -85,B 0,C 180,E1 -13505.759,E2 -13505.759} C_VEL
LIN {X 0,Y 358.156,Z 474.561,A -85,B 0,C 180,E1 -13506.762,E2 -13506.762} C_VEL
LIN {X 0,Y 357.207,Z 482.08,A -85,B 0,C 180,E1 -13507.917,E2 -13507.917} C_VEL
LIN {X 0,Y 356.235,Z 490.203,A -85,B 0,C 180,E1 -13509.471,E2 -13509.471} C_VEL
LIN {X 0,Y 355.51,Z 495.733,A -85,B 0,C 180,E1 -13510.825,E2 -13510.825} C_VEL
LIN {X 0,Y 354.953,Z 499.695,A -85,B 0,C 180,E1 -13512,E2 -13512} C_VEL
LIN {X 0,Y 354.352,Z 504.19,A -85,B 0,C 180,E1 -13513.769,E2 -13513.769} C_VEL
LIN {X 0,Y 354.007,Z 506.48,A -85,B 0,C 180,E1 -13514.957,E2 -13514.957} C_VEL
LIN {X 0,Y 353.733,Z 508.141,A -85,B 0,C 180,E1 -13516.151,E2 -13516.151} C_VEL
LIN {X 0,Y 353.521,Z 509.198,A -85,B 0,C 180,E1 -13517.41,E2 -13517.41} C_VEL
LIN {X 0,Y 353.369,Z 509.602,A -85,B 0,C 180,E1 -13518.556,E2 -13518.556} C_VEL
LIN {X 0,Y 353.271,Z 509.503,A -85,B 0,C 180,E1 -13519.768,E2 -13519.768} C_VEL
LIN {X 0,Y 353.269,Z 508.841,A -85,B 0,C 180,E1 -13520.984,E2 -13520.984} C_VEL
LIN {X 0,Y 353.354,Z 507.59,A -85,B 0,C 180,E1 -13522.204,E2 -13522.204} C_VEL
LIN {X 0,Y 353.527,Z 504.765,A -85,B 0,C 180,E1 -13523.878,E2 -13523.878} C_VEL
LIN {X 0,Y 353.727,Z 501.442,A -85,B 0,C 180,E1 -13525.289,E2 -13525.289} C_VEL
LIN {X 0,Y 353.956,Z 497.159,A -85,B 0,C 180,E1 -13526.69,E2 -13526.69} C_VEL
LIN {X 0,Y 354.319,Z 491.689,A -85,B 0,C 180,E1 -13528.106,E2 -13528.106} C_VEL
LIN {X 0,Y 354.722,Z 485.824,A -85,B 0,C 180,E1 -13529.342,E2 -13529.342} C_VEL
LIN {X 0,Y 355.101,Z 480.369,A -85,B 0,C 180,E1 -13530.311,E2 -13530.311} C_VEL
LIN {X 0,Y 355.601,Z 473.236,A -85,B 0,C 180,E1 -13531.377,E2 -13531.377} C_VEL
LIN {X 0,Y 356.121,Z 465.257,A -85,B 0,C 180,E1 -13532.366,E2 -13532.366} C_VEL
LIN {X 0,Y 356.605,Z 457.56,A -85,B 0,C 180,E1 -13533.155,E2 -13533.155} C_VEL
LIN {X 0,Y 357.04,Z 448.892,A -85,B 0,C 180,E1 -13533.886,E2 -13533.886} C_VEL
LIN {X 0,Y 357.51,Z 439.275,A -85,B 0,C 180,E1 -13534.524,E2 -13534.524} C_VEL
LIN {X 0,Y 357.913,Z 427.587,A -85,B 0,C 180,E1 -13535.098,E2 -13535.098} C_VEL
LIN {X 0,Y 358.333,Z 411.204,A -85,B 0,C 180,E1 -13535.567,E2 -13535.567} C_VEL
LIN {X 0,Y 359.231,Z 363.177,A -85,B 0,C 180,E1 -13536.782,E2 -13536.782} C_VEL
LIN {X 0,Y 356.141,Z 339.614,A -85,B 0,C 180,E1 -13537.545,E2 -13537.545} C_VEL
LIN {X 0,Y 357.332,Z 322.076,A -85,B 0,C 180,E1 -13541.639,E2 -13541.639} C_VEL
LIN {X 0,Y 357.958,Z 313.023,A -85,B 0,C 180,E1 -13543.795,E2 -13543.795} C_VEL
LIN {X 0,Y 356.226,Z 303.176,A -85,B 0,C 180,E1 -13546.331,E2 -13546.331} C_VEL
LIN {X 0,Y 354.802,Z 296.288,A -85,B 0,C 180,E1 -13548.183,E2 -13548.183} C_VEL
LIN {X 0,Y 354.79,Z 296.288,A -85,B 0,C 180,E1 -13552.117,E2 -13552.117} C_VEL
LIN {X 0,Y 354.806,Z 296.285,A -85,B 0,C 180,E1 -13554.941,E2 -13554.941} C_VEL
LIN {X 0,Y 354.79,Z 296.288,A -85,B 0,C 180,E1 -13558.407,E2 -13558.407} C_VEL
LIN {X 0,Y 354.79,Z 296.288,A -85,B 0,C 180,E1 -13561.614,E2 -13561.614} C_VEL
LIN {X 0,Y 354.804,Z 296.285,A -85,B 0,C 180,E1 -13565.42,E2 -13565.42} C_VEL
LIN {X 0,Y 354.826,Z 296.283,A -85,B 0,C 180,E1 -13569.113,E2 -13569.113} C_VEL
LIN {X 0,Y 354.884,Z 296.282,A -85,B 0,C 180,E1 -13572.719,E2 -13572.719} C_VEL
LIN {X 0,Y 354.957,Z 296.266,A -85,B 0,C 180,E1 -13576.254,E2 -13576.254} C_VEL
LIN {X 0,Y 354.959,Z 296.267,A -85,B 0,C 180,E1 -13579.734,E2 -13579.734} C_VEL
LIN {X 0,Y 355.09,Z 296.254,A -85,B 0,C 180,E1 -13583.178,E2 -13583.178} C_VEL
LIN {X 0,Y 355.223,Z 296.238,A -85,B 0,C 180,E1 -13587.73,E2 -13587.73} C_VEL
LIN {X 0,Y 355.148,Z 296.243,A -85,B 0,C 180,E1 -13591.131,E2 -13591.131} C_VEL
LIN {X 0,Y 355.222,Z 296.235,A -85,B 0,C 180,E1 -13592.265,E2 -13592.265} C_VEL
LIN {X 0,Y 355.086,Z 296.25,A -85,B 0,C 180,E1 -13596.817,E2 -13596.817} C_VEL
LIN {X 0,Y 354.953,Z 296.273,A -85,B 0,C 180,E1 -13600.261,E2 -13600.261} C_VEL
LIN {X 0,Y 354.941,Z 296.269,A -85,B 0,C 180,E1 -13604.015,E2 -13604.015} C_VEL
LIN {X 0,Y 354.886,Z 296.275,A -85,B 0,C 180,E1 -13608.088,E2 -13608.088} C_VEL
LIN {X 0,Y 354.801,Z 296.285,A -85,B 0,C 180,E1 -13612.103,E2 -13612.103} C_VEL
LIN {X 0,Y 354.84,Z 296.281,A -85,B 0,C 180,E1 -13614.573,E2 -13614.573} C_VEL
LIN {X 0,Y 354.783,Z 296.287,A -85,B 0,C 180,E1 -13616.452,E2 -13616.452} C_VEL
LIN {X 0,Y 354.111,Z 296.377,A -85,B 0,C 180,E1 -13617.4,E2 -13617.4} C_VEL
LIN {X 0,Y 351.224,Z 296.733,A -85,B 0,C 180,E1 -13618.941,E2 -13618.941} C_VEL
LIN {X 0,Y 348.796,Z 297.034,A -85,B 0,C 180,E1 -13620.189,E2 -13620.189} C_VEL
LIN {X 0,Y 347.783,Z 297.162,A -85,B 0,C 180,E1 -13621.155,E2 -13621.155} C_VEL
LIN {X 0,Y 347.717,Z 297.17,A -85,B 0,C 180,E1 -13621.482,E2 -13621.482} C_VEL
LIN {X 0,Y 347.728,Z 297.167,A -85,B 0,C 180,E1 -13624.459,E2 -13624.459} C_VEL
LIN {X 0,Y 347.752,Z 297.169,A -85,B 0,C 180,E1 -13627.983,E2 -13627.983} C_VEL
LIN {X 0,Y 347.724,Z 297.17,A -85,B 0,C 180,E1 -13631.826,E2 -13631.826} C_VEL
LIN {X 0,Y 347.678,Z 297.173,A -85,B 0,C 180,E1 -13635.022,E2 -13635.022} C_VEL
LIN {X 0,Y 347.721,Z 297.173,A -85,B 0,C 180,E1 -13638.393,E2 -13638.393} C_VEL
LIN {X 0,Y 347.74,Z 297.165,A -85,B 0,C 180,E1 -13642.007,E2 -13642.007} C_VEL
LIN {X 0,Y 347.708,Z 297.17,A -85,B 0,C 180,E1 -13645.531,E2 -13645.531} C_VEL
LIN {X 0,Y 347.727,Z 297.168,A -85,B 0,C 180,E1 -13649.649,E2 -13649.649} C_VEL
LIN {X 0,Y 347.812,Z 297.157,A -85,B 0,C 180,E1 -13652.741,E2 -13652.741} C_VEL
LIN {X 0,Y 347.743,Z 297.165,A -85,B 0,C 180,E1 -13656.158,E2 -13656.158} C_VEL
LIN {X 0,Y 347.732,Z 297.171,A -85,B 0,C 180,E1 -13659.904,E2 -13659.904} C_VEL
LIN {X 0,Y 347.784,Z 297.162,A -85,B 0,C 180,E1 -13663.565,E2 -13663.565} C_VEL
LIN {X 0,Y 347.844,Z 297.152,A -85,B 0,C 180,E1 -13667.158,E2 -13667.158} C_VEL
LIN {X 0,Y 347.897,Z 297.148,A -85,B 0,C 180,E1 -13670.699,E2 -13670.699} C_VEL
LIN {X 0,Y 348.042,Z 297.128,A -85,B 0,C 180,E1 -13673.04,E2 -13673.04} C_VEL
LIN {X 0,Y 348.164,Z 297.112,A -85,B 0,C 180,E1 -13677.686,E2 -13677.686} C_VEL
LIN {X 0,Y 348.274,Z 297.098,A -85,B 0,C 180,E1 -13679.999,E2 -13679.999} C_VEL
LIN {X 0,Y 348.157,Z 297.113,A -85,B 0,C 180,E1 -13682.313,E2 -13682.313} C_VEL
LIN {X 0,Y 348.041,Z 297.13,A -85,B 0,C 180,E1 -13686.958,E2 -13686.958} C_VEL
LIN {X 0,Y 347.88,Z 297.147,A -85,B 0,C 180,E1 -13690.475,E2 -13690.475} C_VEL
LIN {X 0,Y 347.852,Z 297.153,A -85,B 0,C 180,E1 -13694.151,E2 -13694.151} C_VEL
LIN {X 0,Y 347.825,Z 297.157,A -85,B 0,C 180,E1 -13698.282,E2 -13698.282} C_VEL
LIN {X 0,Y 347.731,Z 297.167,A -85,B 0,C 180,E1 -13701.632,E2 -13701.632} C_VEL
LIN {X 0,Y 347.767,Z 297.162,A -85,B 0,C 180,E1 -13705.111,E2 -13705.111} C_VEL
LIN {X 0,Y 347.759,Z 297.163,A -85,B 0,C 180,E1 -13707.698,E2 -13707.698} C_VEL
LIN {X 0,Y 347.7,Z 297.169,A -85,B 0,C 180,E1 -13711.703,E2 -13711.703} C_VEL
LIN {X 0,Y 347.706,Z 297.171,A -85,B 0,C 180,E1 -13714.468,E2 -13714.468} C_VEL
LIN {X 0,Y 347.735,Z 297.165,A -85,B 0,C 180,E1 -13717.992,E2 -13717.992} C_VEL
LIN {X 0,Y 347.715,Z 297.169,A -85,B 0,C 180,E1 -13721.835,E2 -13721.835} C_VEL
LIN {X 0,Y 347.672,Z 297.175,A -85,B 0,C 180,E1 -13725.032,E2 -13725.032} C_VEL
LIN {X 0,Y 347.721,Z 297.168,A -85,B 0,C 180,E1 -13728.402,E2 -13728.402} C_VEL
LIN {X 0,Y 347.737,Z 297.17,A -85,B 0,C 180,E1 -13732.018,E2 -13732.018} C_VEL
LIN {X 0,Y 347.719,Z 297.169,A -85,B 0,C 180,E1 -13735.54,E2 -13735.54} C_VEL
LIN {X 0,Y 347.79,Z 297.203,A -85,B 0,C 180,E1 -13739.031,E2 -13739.031} C_VEL
LIN {X 0,Y 351.008,Z 311.851,A -85,B 0,C 180,E1 -13742.354,E2 -13742.354} C_VEL
LIN {X 0,Y 352.861,Z 320.891,A -85,B 0,C 180,E1 -13744.335,E2 -13744.335} C_VEL
LIN {X 0,Y 352.407,Z 327.027,A -85,B 0,C 180,E1 -13745.561,E2 -13745.561} C_VEL
LIN {X 0,Y 350.62,Z 344.349,A -85,B 0,C 180,E1 -13748.974,E2 -13748.974} C_VEL
LIN {X 0,Y 353.557,Z 372.519,A -85,B 0,C 180,E1 -13749.795,E2 -13749.795} C_VEL
LIN {X 0,Y 352.013,Z 447.796,A -85,B 0,C 180,E1 -13751.564,E2 -13751.564} C_VEL
LIN {X 0,Y 351.643,Z 457.678,A -85,B 0,C 180,E1 -13751.92,E2 -13751.92} C_VEL
LIN {X 0,Y 351.123,Z 466.989,A -85,B 0,C 180,E1 -13752.382,E2 -13752.382} C_VEL
LIN {X 0,Y 350.564,Z 475.972,A -85,B 0,C 180,E1 -13752.955,E2 -13752.955} C_VEL
LIN {X 0,Y 349.843,Z 486.536,A -85,B 0,C 180,E1 -13753.819,E2 -13753.819} C_VEL
LIN {X 0,Y 349.15,Z 496.442,A -85,B 0,C 180,E1 -13754.834,E2 -13754.834} C_VEL
LIN {X 0,Y 348.517,Z 504.492,A -85,B 0,C 180,E1 -13755.827,E2 -13755.827} C_VEL
LIN {X 0,Y 347.934,Z 511.677,A -85,B 0,C 180,E1 -13756.869,E2 -13756.869} C_VEL
LIN {X 0,Y 347.359,Z 519.986,A -85,B 0,C 180,E1 -13758.331,E2 -13758.331} C_VEL
LIN {X 0,Y 346.879,Z 526.838,A -85,B 0,C 180,E1 -13759.792,E2 -13759.792} C_VEL
LIN {X 0,Y 346.592,Z 532.51,A -85,B 0,C 180,E1 -13761.256,E2 -13761.256} C_VEL
LIN {X 0,Y 346.445,Z 536.377,A -85,B 0,C 180,E1 -13762.426,E2 -13762.426} C_VEL
LIN {X 0,Y 346.283,Z 540.944,A -85,B 0,C 180,E1 -13764.179,E2 -13764.179} C_VEL
LIN {X 0,Y 346.343,Z 543.294,A -85,B 0,C 180,E1 -13765.347,E2 -13765.347} C_VEL
LIN {X 0,Y 346.341,Z 546.649,A -85,B 0,C 180,E1 -13767.677,E2 -13767.677} C_VEL
LIN {X 0,Y 346.403,Z 547.593,A -85,B 0,C 180,E1 -13768.84,E2 -13768.84} C_VEL
LIN {X 0,Y 346.348,Z 548.248,A -85,B 0,C 180,E1 -13771.165,E2 -13771.165} C_VEL
LIN {X 0,Y 346.197,Z 547.031,A -85,B 0,C 180,E1 -13773.494,E2 -13773.494} C_VEL
LIN {X 0,Y 346.209,Z 545.896,A -85,B 0,C 180,E1 -13774.659,E2 -13774.659} C_VEL
LIN {X 0,Y 346.239,Z 543.96,A -85,B 0,C 180,E1 -13775.958,E2 -13775.958} C_VEL
LIN {X 0,Y 346.483,Z 539.477,A -85,B 0,C 180,E1 -13778.164,E2 -13778.164} C_VEL
LIN {X 0,Y 346.88,Z 534.552,A -85,B 0,C 180,E1 -13779.918,E2 -13779.918} C_VEL
LIN {X 0,Y 347.516,Z 528.326,A -85,B 0,C 180,E1 -13781.669,E2 -13781.669} C_VEL
LIN {X 0,Y 348.334,Z 522.014,A -85,B 0,C 180,E1 -13783.12,E2 -13783.12} C_VEL
LIN {X 0,Y 349.198,Z 514.404,A -85,B 0,C 180,E1 -13784.571,E2 -13784.571} C_VEL
LIN {X 0,Y 350.26,Z 506.164,A -85,B 0,C 180,E1 -13785.866,E2 -13785.866} C_VEL
LIN {X 0,Y 351.44,Z 497.374,A -85,B 0,C 180,E1 -13787.006,E2 -13787.006} C_VEL
LIN {X 0,Y 352.359,Z 489.604,A -85,B 0,C 180,E1 -13787.859,E2 -13787.859} C_VEL
LIN {X 0,Y 353.425,Z 480.26,A -85,B 0,C 180,E1 -13788.703,E2 -13788.703} C_VEL
LIN {X 0,Y 354.438,Z 469.509,A -85,B 0,C 180,E1 -13789.474,E2 -13789.474} C_VEL
LIN {X 0,Y 355.202,Z 459.53,A -85,B 0,C 180,E1 -13790.032,E2 -13790.032} C_VEL
LIN {X 0,Y 355.933,Z 448.243,A -85,B 0,C 180,E1 -13790.479,E2 -13790.479} C_VEL
LIN {X 0,Y 356.784,Z 421.71,A -85,B 0,C 180,E1 -13791.157,E2 -13791.157} C_VEL
LIN {X 0,Y 358.351,Z 371.568,A -85,B 0,C 180,E1 -13792.407,E2 -13792.407} C_VEL
LIN {X 0,Y 355.95,Z 353.987,A -85,B 0,C 180,E1 -13793.122,E2 -13793.122} C_VEL
LIN {X 0,Y 353.973,Z 343.093,A -85,B 0,C 180,E1 -13793.655,E2 -13793.655} C_VEL
LIN {X 0,Y 355.685,Z 327.484,A -85,B 0,C 180,E1 -13796.553,E2 -13796.553} C_VEL
LIN {X 0,Y 353.961,Z 318.291,A -85,B 0,C 180,E1 -13798.618,E2 -13798.618} C_VEL
LIN {X 0,Y 351.296,Z 308.293,A -85,B 0,C 180,E1 -13801.065,E2 -13801.065} C_VEL
LIN {X 0,Y 347.74,Z 297.17,A -85,B 0,C 180,E1 -13804.089,E2 -13804.089} C_VEL
LIN {X 0,Y 347.753,Z 297.172,A -85,B 0,C 180,E1 -13807.32,E2 -13807.32} C_VEL
LIN {X 0,Y 347.723,Z 297.175,A -85,B 0,C 180,E1 -13810.296,E2 -13810.296} C_VEL
LIN {X 0,Y 347.713,Z 297.173,A -85,B 0,C 180,E1 -13813.407,E2 -13813.407} C_VEL
LIN {X 0,Y 347.715,Z 297.173,A -85,B 0,C 180,E1 -13816.685,E2 -13816.685} C_VEL
LIN {X 0,Y 347.744,Z 297.165,A -85,B 0,C 180,E1 -13820.171,E2 -13820.171} C_VEL
LIN {X 0,Y 347.755,Z 297.164,A -85,B 0,C 180,E1 -13823.934,E2 -13823.934} C_VEL
LIN {X 0,Y 347.717,Z 297.161,A -85,B 0,C 180,E1 -13826.927,E2 -13826.927} C_VEL
LIN {X 0,Y 347.788,Z 297.157,A -85,B 0,C 180,E1 -13830.989,E2 -13830.989} C_VEL
LIN {X 0,Y 347.813,Z 297.156,A -85,B 0,C 180,E1 -13833.607,E2 -13833.607} C_VEL
LIN {X 0,Y 347.78,Z 297.161,A -85,B 0,C 180,E1 -13836.162,E2 -13836.162} C_VEL
LIN {X 0,Y 347.815,Z 297.161,A -85,B 0,C 180,E1 -13839.91,E2 -13839.91} C_VEL
LIN {X 0,Y 347.846,Z 297.155,A -85,B 0,C 180,E1 -13842.359,E2 -13842.359} C_VEL
LIN {X 0,Y 347.878,Z 297.151,A -85,B 0,C 180,E1 -13845.971,E2 -13845.971} C_VEL
LIN {X 0,Y 347.911,Z 297.152,A -85,B 0,C 180,E1 -13850.114,E2 -13850.114} C_VEL
LIN {X 0,Y 347.911,Z 297.156,A -85,B 0,C 180,E1 -13850.261,E2 -13850.261} C_VEL
LIN {X 0,Y 351.577,Z 308.151,A -85,B 0,C 180,E1 -13853.112,E2 -13853.112} C_VEL
LIN {X 0,Y 354.286,Z 319.403,A -85,B 0,C 180,E1 -13855.702,E2 -13855.702} C_VEL
LIN {X 0,Y 352.98,Z 336.476,A -85,B 0,C 180,E1 -13858.86,E2 -13858.86} C_VEL
LIN {X 0,Y 352.839,Z 338.42,A -85,B 0,C 180,E1 -13859.216,E2 -13859.216} C_VEL
LIN {X 0,Y 356.712,Z 358.028,A -85,B 0,C 180,E1 -13860.248,E2 -13860.248} C_VEL
LIN {X 0,Y 358.056,Z 367.345,A -85,B 0,C 180,E1 -13860.668,E2 -13860.668} C_VEL
LIN {X 0,Y 355.594,Z 425.888,A -85,B 0,C 180,E1 -13862.372,E2 -13862.372} C_VEL
LIN {X 0,Y 354.903,Z 437.948,A -85,B 0,C 180,E1 -13862.909,E2 -13862.909} C_VEL
LIN {X 0,Y 354.003,Z 449.847,A -85,B 0,C 180,E1 -13863.7,E2 -13863.7} C_VEL
LIN {X 0,Y 353.109,Z 459.721,A -85,B 0,C 180,E1 -13864.567,E2 -13864.567} C_VEL
LIN {X 0,Y 352.267,Z 468.04,A -85,B 0,C 180,E1 -13865.471,E2 -13865.471} C_VEL
LIN {X 0,Y 351.248,Z 476.629,A -85,B 0,C 180,E1 -13866.607,E2 -13866.607} C_VEL
LIN {X 0,Y 350.118,Z 485.454,A -85,B 0,C 180,E1 -13868.078,E2 -13868.078} C_VEL
LIN {X 0,Y 349.181,Z 492.304,A -85,B 0,C 180,E1 -13869.541,E2 -13869.541} C_VEL
LIN {X 0,Y 348.645,Z 495.964,A -85,B 0,C 180,E1 -13870.453,E2 -13870.453} C_VEL
LIN {X 0,Y 348.059,Z 499.929,A -85,B 0,C 180,E1 -13871.65,E2 -13871.65} C_VEL
LIN {X 0,Y 347.59,Z 503.127,A -85,B 0,C 180,E1 -13872.851,E2 -13872.851} C_VEL
LIN {X 0,Y 347.218,Z 505.667,A -85,B 0,C 180,E1 -13874.058,E2 -13874.058} C_VEL
LIN {X 0,Y 346.864,Z 507.632,A -85,B 0,C 180,E1 -13875.273,E2 -13875.273} C_VEL
LIN {X 0,Y 346.582,Z 509.036,A -85,B 0,C 180,E1 -13876.493,E2 -13876.493} C_VEL
LIN {X 0,Y 346.392,Z 509.886,A -85,B 0,C 180,E1 -13877.719,E2 -13877.719} C_VEL
LIN {X 0,Y 346.256,Z 510.124,A -85,B 0,C 180,E1 -13878.951,E2 -13878.951} C_VEL
LIN {X 0,Y 346.188,Z 509.188,A -85,B 0,C 180,E1 -13880.965,E2 -13880.965} C_VEL
LIN {X 0,Y 346.373,Z 506.19,A -85,B 0,C 180,E1 -13883.308,E2 -13883.308} C_VEL
LIN {X 0,Y 346.639,Z 502.069,A -85,B 0,C 180,E1 -13885.2,E2 -13885.2} C_VEL
LIN {X 0,Y 346.949,Z 496.639,A -85,B 0,C 180,E1 -13886.97,E2 -13886.97} C_VEL
LIN {X 0,Y 347.317,Z 491.058,A -85,B 0,C 180,E1 -13888.394,E2 -13888.394} C_VEL
LIN {X 0,Y 347.872,Z 483.526,A -85,B 0,C 180,E1 -13889.938,E2 -13889.938} C_VEL
LIN {X 0,Y 348.448,Z 475.127,A -85,B 0,C 180,E1 -13891.29,E2 -13891.29} C_VEL
LIN {X 0,Y 349.026,Z 466.812,A -85,B 0,C 180,E1 -13892.372,E2 -13892.372} C_VEL
LIN {X 0,Y 349.534,Z 458.884,A -85,B 0,C 180,E1 -13893.224,E2 -13893.224} C_VEL
LIN {X 0,Y 350.01,Z 449.596,A -85,B 0,C 180,E1 -13894.037,E2 -13894.037} C_VEL
LIN {X 0,Y 350.44,Z 441.351,A -85,B 0,C 180,E1 -13894.612,E2 -13894.612} C_VEL
LIN {X 0,Y 350.839,Z 431.2,A -85,B 0,C 180,E1 -13895.156,E2 -13895.156} C_VEL
LIN {X 0,Y 351.154,Z 419.431,A -85,B 0,C 180,E1 -13895.59,E2 -13895.59} C_VEL
LIN {X 0,Y 352.361,Z 364.174,A -85,B 0,C 180,E1 -13897.022,E2 -13897.022} C_VEL
LIN {X 0,Y 349.174,Z 339.669,A -85,B 0,C 180,E1 -13897.826,E2 -13897.826} C_VEL
LIN {X 0,Y 350.363,Z 322.99,A -85,B 0,C 180,E1 -13901.784,E2 -13901.784} C_VEL
LIN {X 0,Y 350.984,Z 314.331,A -85,B 0,C 180,E1 -13903.878,E2 -13903.878} C_VEL
LIN {X 0,Y 349.283,Z 304.628,A -85,B 0,C 180,E1 -13906.417,E2 -13906.417} C_VEL
LIN {X 0,Y 347.751,Z 297.166,A -85,B 0,C 180,E1 -13908.493,E2 -13908.493} C_VEL
LIN {X 0,Y 347.752,Z 297.163,A -85,B 0,C 180,E1 -13912.679,E2 -13912.679} C_VEL
LIN {X 0,Y 347.748,Z 297.169,A -85,B 0,C 180,E1 -13915.958,E2 -13915.958} C_VEL
LIN {X 0,Y 347.736,Z 297.168,A -85,B 0,C 180,E1 -13919.651,E2 -13919.651} C_VEL
LIN {X 0,Y 347.734,Z 297.166,A -85,B 0,C 180,E1 -13923.6,E2 -13923.6} C_VEL
LIN {X 0,Y 347.751,Z 297.168,A -85,B 0,C 180,E1 -13926.159,E2 -13926.159} C_VEL
LIN {X 0,Y 347.784,Z 297.16,A -85,B 0,C 180,E1 -13929.907,E2 -13929.907} C_VEL
LIN {X 0,Y 347.847,Z 297.154,A -85,B 0,C 180,E1 -13932.358,E2 -13932.358} C_VEL
LIN {X 0,Y 347.903,Z 297.144,A -85,B 0,C 180,E1 -13935.97,E2 -13935.97} C_VEL
LIN {X 0,Y 347.899,Z 297.147,A -85,B 0,C 180,E1 -13939.523,E2 -13939.523} C_VEL
LIN {X 0,Y 348.057,Z 297.129,A -85,B 0,C 180,E1 -13943.04,E2 -13943.04} C_VEL
LIN {X 0,Y 348.184,Z 297.115,A -85,B 0,C 180,E1 -13947.684,E2 -13947.684} C_VEL
LIN {X 0,Y 348.119,Z 297.118,A -85,B 0,C 180,E1 -13951.154,E2 -13951.154} C_VEL
LIN {X 0,Y 348.184,Z 297.112,A -85,B 0,C 180,E1 -13952.311,E2 -13952.311} C_VEL
LIN {X 0,Y 348.054,Z 297.126,A -85,B 0,C 180,E1 -13956.956,E2 -13956.956} C_VEL
LIN {X 0,Y 347.894,Z 297.151,A -85,B 0,C 180,E1 -13960.472,E2 -13960.472} C_VEL
LIN {X 0,Y 347.898,Z 297.148,A -85,B 0,C 180,E1 -13964.146,E2 -13964.146} C_VEL
LIN {X 0,Y 347.825,Z 297.156,A -85,B 0,C 180,E1 -13968.255,E2 -13968.255} C_VEL
LIN {X 0,Y 347.758,Z 297.163,A -85,B 0,C 180,E1 -13971.62,E2 -13971.62} C_VEL
LIN {X 0,Y 347.76,Z 297.169,A -85,B 0,C 180,E1 -13975.107,E2 -13975.107} C_VEL
LIN {X 0,Y 347.725,Z 297.169,A -85,B 0,C 180,E1 -13977.696,E2 -13977.696} C_VEL
LIN {X 0,Y 347.725,Z 297.167,A -85,B 0,C 180,E1 -13980.344,E2 -13980.344} C_VEL
LIN {X 0,Y 347.717,Z 297.17,A -85,B 0,C 180,E1 -13981.482,E2 -13981.482} C_VEL
LIN {X 0,Y 347.093,Z 297.255,A -85,B 0,C 180,E1 -13982.449,E2 -13982.449} C_VEL
LIN {X 0,Y 344.256,Z 297.61,A -85,B 0,C 180,E1 -13984.022,E2 -13984.022} C_VEL
LIN {X 0,Y 341.823,Z 297.908,A -85,B 0,C 180,E1 -13985.296,E2 -13985.296} C_VEL
LIN {X 0,Y 340.774,Z 298.035,A -85,B 0,C 180,E1 -13986.281,E2 -13986.281} C_VEL
LIN {X 0,Y 340.687,Z 298.044,A -85,B 0,C 180,E1 -13986.615,E2 -13986.615} C_VEL
LIN {X 0,Y 340.677,Z 298.048,A -85,B 0,C 180,E1 -13989.748,E2 -13989.748} C_VEL
LIN {X 0,Y 340.651,Z 298.048,A -85,B 0,C 180,E1 -13992.9,E2 -13992.9} C_VEL
LIN {X 0,Y 340.648,Z 298.049,A -85,B 0,C 180,E1 -13997.09,E2 -13997.09} C_VEL
LIN {X 0,Y 340.669,Z 298.048,A -85,B 0,C 180,E1 -14000.242,E2 -14000.242} C_VEL
LIN {X 0,Y 340.675,Z 298.045,A -85,B 0,C 180,E1 -14003.556,E2 -14003.556} C_VEL
LIN {X 0,Y 340.655,Z 298.047,A -85,B 0,C 180,E1 -14006.148,E2 -14006.148} C_VEL
LIN {X 0,Y 340.737,Z 298.037,A -85,B 0,C 180,E1 -14010.328,E2 -14010.328} C_VEL
LIN {X 0,Y 340.765,Z 298.037,A -85,B 0,C 180,E1 -14013.016,E2 -14013.016} C_VEL
LIN {X 0,Y 340.713,Z 298.045,A -85,B 0,C 180,E1 -14015.634,E2 -14015.634} C_VEL
LIN {X 0,Y 340.67,Z 298.049,A -85,B 0,C 180,E1 -14019.469,E2 -14019.469} C_VEL
LIN {X 0,Y 340.731,Z 298.043,A -85,B 0,C 180,E1 -14021.977,E2 -14021.977} C_VEL
LIN {X 0,Y 340.808,Z 298.031,A -85,B 0,C 180,E1 -14025.714,E2 -14025.714} C_VEL
LIN {X 0,Y 340.825,Z 298.026,A -85,B 0,C 180,E1 -14029.304,E2 -14029.304} C_VEL
LIN {X 0,Y 341.01,Z 298.005,A -85,B 0,C 180,E1 -14032.896,E2 -14032.896} C_VEL
LIN {X 0,Y 341.126,Z 297.989,A -85,B 0,C 180,E1 -14037.638,E2 -14037.638} C_VEL
LIN {X 0,Y 341.225,Z 297.976,A -85,B 0,C 180,E1 -14039.999,E2 -14039.999} C_VEL
LIN {X 0,Y 341.119,Z 297.99,A -85,B 0,C 180,E1 -14042.361,E2 -14042.361} C_VEL
LIN {X 0,Y 341.009,Z 298.008,A -85,B 0,C 180,E1 -14047.103,E2 -14047.103} C_VEL
LIN {X 0,Y 340.822,Z 298.027,A -85,B 0,C 180,E1 -14050.695,E2 -14050.695} C_VEL
LIN {X 0,Y 340.817,Z 298.028,A -85,B 0,C 180,E1 -14054.326,E2 -14054.326} C_VEL
LIN {X 0,Y 340.776,Z 298.034,A -85,B 0,C 180,E1 -14058.46,E2 -14058.46} C_VEL
LIN {X 0,Y 340.677,Z 298.048,A -85,B 0,C 180,E1 -14061.845,E2 -14061.845} C_VEL
LIN {X 0,Y 340.728,Z 298.039,A -85,B 0,C 180,E1 -14065.667,E2 -14065.667} C_VEL
LIN {X 0,Y 340.676,Z 298.049,A -85,B 0,C 180,E1 -14068.325,E2 -14068.325} C_VEL
LIN {X 0,Y 340.651,Z 298.051,A -85,B 0,C 180,E1 -14071.049,E2 -14071.049} C_VEL
LIN {X 0,Y 340.679,Z 298.047,A -85,B 0,C 180,E1 -14075.283,E2 -14075.283} C_VEL
LIN {X 0,Y 340.672,Z 298.046,A -85,B 0,C 180,E1 -14078.389,E2 -14078.389} C_VEL
LIN {X 0,Y 340.664,Z 298.046,A -85,B 0,C 180,E1 -14082.049,E2 -14082.049} C_VEL
LIN {X 0,Y 340.621,Z 298.052,A -85,B 0,C 180,E1 -14086.231,E2 -14086.231} C_VEL
LIN {X 0,Y 340.649,Z 298.055,A -85,B 0,C 180,E1 -14089.76,E2 -14089.76} C_VEL
LIN {X 0,Y 340.676,Z 298.045,A -85,B 0,C 180,E1 -14093.262,E2 -14093.262} C_VEL
LIN {X 0,Y 340.67,Z 298.052,A -85,B 0,C 180,E1 -14096.158,E2 -14096.158} C_VEL
LIN {X 0,Y 340.726,Z 298.125,A -85,B 0,C 180,E1 -14098.705,E2 -14098.705} C_VEL
LIN {X 0,Y 343.502,Z 310.578,A -85,B 0,C 180,E1 -14101.614,E2 -14101.614} C_VEL
LIN {X 0,Y 345.821,Z 321.702,A -85,B 0,C 180,E1 -14104.107,E2 -14104.107} C_VEL
LIN {X 0,Y 345.885,Z 324.756,A -85,B 0,C 180,E1 -14104.747,E2 -14104.747} C_VEL
LIN {X 0,Y 343.684,Z 344.17,A -85,B 0,C 180,E1 -14108.654,E2 -14108.654} C_VEL
LIN {X 0,Y 346.64,Z 373.255,A -85,B 0,C 180,E1 -14109.541,E2 -14109.541} C_VEL
LIN {X 0,Y 345.038,Z 448.486,A -85,B 0,C 180,E1 -14111.37,E2 -14111.37} C_VEL
LIN {X 0,Y 344.654,Z 458.024,A -85,B 0,C 180,E1 -14111.733,E2 -14111.733} C_VEL
LIN {X 0,Y 344.105,Z 467.762,A -85,B 0,C 180,E1 -14112.241,E2 -14112.241} C_VEL
LIN {X 0,Y 343.48,Z 477.44,A -85,B 0,C 180,E1 -14112.899,E2 -14112.899} C_VEL
LIN {X 0,Y 342.85,Z 486.15,A -85,B 0,C 180,E1 -14113.633,E2 -14113.633} C_VEL
LIN {X 0,Y 342.108,Z 495.999,A -85,B 0,C 180,E1 -14114.66,E2 -14114.66} C_VEL
LIN {X 0,Y 341.452,Z 504.286,A -85,B 0,C 180,E1 -14115.704,E2 -14115.704} C_VEL
LIN {X 0,Y 340.801,Z 512.179,A -85,B 0,C 180,E1 -14116.893,E2 -14116.893} C_VEL
LIN {X 0,Y 340.373,Z 518.905,A -85,B 0,C 180,E1 -14118.088,E2 -14118.088} C_VEL
LIN {X 0,Y 339.84,Z 525.88,A -85,B 0,C 180,E1 -14119.578,E2 -14119.578} C_VEL
LIN {X 0,Y 339.521,Z 531.66,A -85,B 0,C 180,E1 -14121.072,E2 -14121.072} C_VEL
LIN {X 0,Y 339.327,Z 537.197,A -85,B 0,C 180,E1 -14122.865,E2 -14122.865} C_VEL
LIN {X 0,Y 339.2,Z 540.947,A -85,B 0,C 180,E1 -14124.395,E2 -14124.395} C_VEL
LIN {X 0,Y 339.273,Z 542.633,A -85,B 0,C 180,E1 -14125.25,E2 -14125.25} C_VEL
LIN {X 0,Y 339.246,Z 546.129,A -85,B 0,C 180,E1 -14127.628,E2 -14127.628} C_VEL
LIN {X 0,Y 339.341,Z 547.082,A -85,B 0,C 180,E1 -14128.816,E2 -14128.816} C_VEL
LIN {X 0,Y 339.327,Z 547.637,A -85,B 0,C 180,E1 -14130.002,E2 -14130.002} C_VEL
LIN {X 0,Y 339.252,Z 547.849,A -85,B 0,C 180,E1 -14131.189,E2 -14131.189} C_VEL
LIN {X 0,Y 339.118,Z 546.704,A -85,B 0,C 180,E1 -14133.567,E2 -14133.567} C_VEL
LIN {X 0,Y 339.105,Z 545.599,A -85,B 0,C 180,E1 -14134.757,E2 -14134.757} C_VEL
LIN {X 0,Y 339.193,Z 542.984,A -85,B 0,C 180,E1 -14136.545,E2 -14136.545} C_VEL
LIN {X 0,Y 339.423,Z 539.319,A -85,B 0,C 180,E1 -14138.335,E2 -14138.335} C_VEL
LIN {X 0,Y 339.862,Z 534.501,A -85,B 0,C 180,E1 -14140.125,E2 -14140.125} C_VEL
LIN {X 0,Y 340.536,Z 528.357,A -85,B 0,C 180,E1 -14141.912,E2 -14141.912} C_VEL
LIN {X 0,Y 341.406,Z 522.124,A -85,B 0,C 180,E1 -14143.392,E2 -14143.392} C_VEL
LIN {X 0,Y 342.276,Z 514.948,A -85,B 0,C 180,E1 -14144.811,E2 -14144.811} C_VEL
LIN {X 0,Y 343.445,Z 506.459,A -85,B 0,C 180,E1 -14146.19,E2 -14146.19} C_VEL
LIN {X 0,Y 344.686,Z 497.833,A -85,B 0,C 180,E1 -14147.35,E2 -14147.35} C_VEL
LIN {X 0,Y 345.821,Z 488.811,A -85,B 0,C 180,E1 -14148.361,E2 -14148.361} C_VEL
LIN {X 0,Y 346.969,Z 479.434,A -85,B 0,C 180,E1 -14149.218,E2 -14149.218} C_VEL
LIN {X 0,Y 347.923,Z 469.807,A -85,B 0,C 180,E1 -14149.93,E2 -14149.93} C_VEL
LIN {X 0,Y 348.796,Z 459.265,A -85,B 0,C 180,E1 -14150.532,E2 -14150.532} C_VEL
LIN {X 0,Y 349.562,Z 448.024,A -85,B 0,C 180,E1 -14150.985,E2 -14150.985} C_VEL
LIN {X 0,Y 350.44,Z 422,A -85,B 0,C 180,E1 -14151.669,E2 -14151.669} C_VEL
LIN {X 0,Y 352.106,Z 372.283,A -85,B 0,C 180,E1 -14152.941,E2 -14152.941} C_VEL
LIN {X 0,Y 349.773,Z 355.08,A -85,B 0,C 180,E1 -14153.682,E2 -14153.682} C_VEL
LIN {X 0,Y 347.527,Z 343.094,A -85,B 0,C 180,E1 -14154.274,E2 -14154.274} C_VEL
LIN {X 0,Y 349.132,Z 329.849,A -85,B 0,C 180,E1 -14156.794,E2 -14156.794} C_VEL
LIN {X 0,Y 347.634,Z 321.54,A -85,B 0,C 180,E1 -14158.694,E2 -14158.694} C_VEL
LIN {X 0,Y 345.062,Z 311.6,A -85,B 0,C 180,E1 -14161.194,E2 -14161.194} C_VEL
LIN {X 0,Y 342.256,Z 302.639,A -85,B 0,C 180,E1 -14163.67,E2 -14163.67} C_VEL
LIN {X 0,Y 340.69,Z 298.049,A -85,B 0,C 180,E1 -14165.034,E2 -14165.034} C_VEL
LIN {X 0,Y 340.701,Z 298.049,A -85,B 0,C 180,E1 -14168.385,E2 -14168.385} C_VEL
LIN {X 0,Y 340.689,Z 298.05,A -85,B 0,C 180,E1 -14172.045,E2 -14172.045} C_VEL
LIN {X 0,Y 340.641,Z 298.054,A -85,B 0,C 180,E1 -14176.226,E2 -14176.226} C_VEL
LIN {X 0,Y 340.694,Z 298.044,A -85,B 0,C 180,E1 -14179.749,E2 -14179.749} C_VEL
LIN {X 0,Y 340.691,Z 298.043,A -85,B 0,C 180,E1 -14183.257,E2 -14183.257} C_VEL
LIN {X 0,Y 340.678,Z 298.044,A -85,B 0,C 180,E1 -14186.152,E2 -14186.152} C_VEL
LIN {X 0,Y 340.758,Z 298.032,A -85,B 0,C 180,E1 -14190.332,E2 -14190.332} C_VEL
LIN {X 0,Y 340.787,Z 298.032,A -85,B 0,C 180,E1 -14193.019,E2 -14193.019} C_VEL
LIN {X 0,Y 340.762,Z 298.038,A -85,B 0,C 180,E1 -14195.639,E2 -14195.639} C_VEL
LIN {X 0,Y 340.758,Z 298.04,A -85,B 0,C 180,E1 -14199.476,E2 -14199.476} C_VEL
LIN {X 0,Y 340.839,Z 298.03,A -85,B 0,C 180,E1 -14201.984,E2 -14201.984} C_VEL
LIN {X 0,Y 340.833,Z 298.029,A -85,B 0,C 180,E1 -14205.716,E2 -14205.716} C_VEL
LIN {X 0,Y 340.851,Z 298.073,A -85,B 0,C 180,E1 -14209.306,E2 -14209.306} C_VEL
LIN {X 0,Y 345.101,Z 310.333,A -85,B 0,C 180,E1 -14212.688,E2 -14212.688} C_VEL
LIN {X 0,Y 347.783,Z 321.572,A -85,B 0,C 180,E1 -14215.364,E2 -14215.364} C_VEL
LIN {X 0,Y 346.636,Z 335.324,A -85,B 0,C 180,E1 -14217.967,E2 -14217.967} C_VEL
LIN {X 0,Y 346.449,Z 338.781,A -85,B 0,C 180,E1 -14218.584,E2 -14218.584} C_VEL
LIN {X 0,Y 350.244,Z 357.405,A -85,B 0,C 180,E1 -14219.613,E2 -14219.613} C_VEL
LIN {X 0,Y 351.795,Z 368.915,A -85,B 0,C 180,E1 -14220.158,E2 -14220.158} C_VEL
LIN {X 0,Y 349.177,Z 427.283,A -85,B 0,C 180,E1 -14221.911,E2 -14221.911} C_VEL
LIN {X 0,Y 348.361,Z 440.176,A -85,B 0,C 180,E1 -14222.53,E2 -14222.53} C_VEL
LIN {X 0,Y 347.587,Z 449.752,A -85,B 0,C 180,E1 -14223.188,E2 -14223.188} C_VEL
LIN {X 0,Y 346.621,Z 459.727,A -85,B 0,C 180,E1 -14224.07,E2 -14224.07} C_VEL
LIN {X 0,Y 345.676,Z 468.31,A -85,B 0,C 180,E1 -14225.017,E2 -14225.017} C_VEL
LIN {X 0,Y 344.627,Z 476.68,A -85,B 0,C 180,E1 -14226.147,E2 -14226.147} C_VEL
LIN {X 0,Y 343.386,Z 485.588,A -85,B 0,C 180,E1 -14227.646,E2 -14227.646} C_VEL
LIN {X 0,Y 342.369,Z 492.564,A -85,B 0,C 180,E1 -14229.155,E2 -14229.155} C_VEL
LIN {X 0,Y 341.671,Z 497.09,A -85,B 0,C 180,E1 -14230.339,E2 -14230.339} C_VEL
LIN {X 0,Y 340.893,Z 501.83,A -85,B 0,C 180,E1 -14231.898,E2 -14231.898} C_VEL
LIN {X 0,Y 340.442,Z 504.794,A -85,B 0,C 180,E1 -14233.126,E2 -14233.126} C_VEL
LIN {X 0,Y 340.07,Z 507.136,A -85,B 0,C 180,E1 -14234.36,E2 -14234.36} C_VEL
LIN {X 0,Y 339.705,Z 508.817,A -85,B 0,C 180,E1 -14235.603,E2 -14235.603} C_VEL
LIN {X 0,Y 339.31,Z 510.341,A -85,B 0,C 180,E1 -14237.688,E2 -14237.688} C_VEL
LIN {X 0,Y 339.146,Z 510.404,A -85,B 0,C 180,E1 -14239.364,E2 -14239.364} C_VEL
LIN {X 0,Y 339.1,Z 509.329,A -85,B 0,C 180,E1 -14241.157,E2 -14241.157} C_VEL
LIN {X 0,Y 339.153,Z 508.612,A -85,B 0,C 180,E1 -14241.901,E2 -14241.901} C_VEL
LIN {X 0,Y 339.355,Z 505.662,A -85,B 0,C 180,E1 -14243.765,E2 -14243.765} C_VEL
LIN {X 0,Y 339.526,Z 502.692,A -85,B 0,C 180,E1 -14245.11,E2 -14245.11} C_VEL
LIN {X 0,Y 339.806,Z 497.934,A -85,B 0,C 180,E1 -14246.734,E2 -14246.734} C_VEL
LIN {X 0,Y 340.159,Z 493.071,A -85,B 0,C 180,E1 -14248.061,E2 -14248.061} C_VEL
LIN {X 0,Y 340.535,Z 487.308,A -85,B 0,C 180,E1 -14249.352,E2 -14249.352} C_VEL
LIN {X 0,Y 340.973,Z 481.509,A -85,B 0,C 180,E1 -14250.44,E2 -14250.44} C_VEL
LIN {X 0,Y 341.544,Z 473.733,A -85,B 0,C 180,E1 -14251.65,E2 -14251.65} C_VEL
LIN {X 0,Y 342.092,Z 465.232,A -85,B 0,C 180,E1 -14252.736,E2 -14252.736} C_VEL
LIN {X 0,Y 342.668,Z 456.686,A -85,B 0,C 180,E1 -14253.626,E2 -14253.626} C_VEL
LIN {X 0,Y 343.317,Z 445.856,A -85,B 0,C 180,E1 -14254.527,E2 -14254.527} C_VEL
LIN {X 0,Y 343.734,Z 434.04,A -85,B 0,C 180,E1 -14255.235,E2 -14255.235} C_VEL
LIN {X 0,Y 344.127,Z 423.87,A -85,B 0,C 180,E1 -14255.66,E2 -14255.66} C_VEL
LIN {X 0,Y 345.476,Z 365.067,A -85,B 0,C 180,E1 -14257.262,E2 -14257.262} C_VEL
LIN {X 0,Y 342.221,Z 339.603,A -85,B 0,C 180,E1 -14258.136,E2 -14258.136} C_VEL
LIN {X 0,Y 343.454,Z 323.288,A -85,B 0,C 180,E1 -14262.08,E2 -14262.08} C_VEL
LIN {X 0,Y 344.029,Z 315.512,A -85,B 0,C 180,E1 -14263.994,E2 -14263.994} C_VEL
LIN {X 0,Y 342.309,Z 305.87,A -85,B 0,C 180,E1 -14266.562,E2 -14266.562} C_VEL
LIN {X 0,Y 340.699,Z 298.046,A -85,B 0,C 180,E1 -14268.768,E2 -14268.768} C_VEL
LIN {X 0,Y 340.715,Z 298.044,A -85,B 0,C 180,E1 -14271.772,E2 -14271.772} C_VEL
LIN {X 0,Y 340.721,Z 298.044,A -85,B 0,C 180,E1 -14275.597,E2 -14275.597} C_VEL
LIN {X 0,Y 340.691,Z 298.043,A -85,B 0,C 180,E1 -14278.955,E2 -14278.955} C_VEL
LIN {X 0,Y 340.711,Z 298.04,A -85,B 0,C 180,E1 -14283.012,E2 -14283.012} C_VEL
LIN {X 0,Y 340.703,Z 298.043,A -85,B 0,C 180,E1 -14286.925,E2 -14286.925} C_VEL
LIN {X 0,Y 340.728,Z 298.044,A -85,B 0,C 180,E1 -14290.729,E2 -14290.729} C_VEL
LIN {X 0,Y 340.821,Z 298.029,A -85,B 0,C 180,E1 -14294.45,E2 -14294.45} C_VEL
LIN {X 0,Y 340.853,Z 298.023,A -85,B 0,C 180,E1 -14298.1,E2 -14298.1} C_VEL
LIN {X 0,Y 340.985,Z 298.008,A -85,B 0,C 180,E1 -14301.703,E2 -14301.703} C_VEL
LIN {X 0,Y 341.016,Z 298.003,A -85,B 0,C 180,E1 -14304.084,E2 -14304.084} C_VEL
LIN {X 0,Y 341.121,Z 297.996,A -85,B 0,C 180,E1 -14307.636,E2 -14307.636} C_VEL
LIN {X 0,Y 341.09,Z 297.994,A -85,B 0,C 180,E1 -14311.178,E2 -14311.178} C_VEL
LIN {X 0,Y 341.12,Z 297.991,A -85,B 0,C 180,E1 -14312.359,E2 -14312.359} C_VEL
LIN {X 0,Y 341.013,Z 298.008,A -85,B 0,C 180,E1 -14315.912,E2 -14315.912} C_VEL
LIN {X 0,Y 340.965,Z 298.014,A -85,B 0,C 180,E1 -14318.353,E2 -14318.353} C_VEL
LIN {X 0,Y 340.847,Z 298.025,A -85,B 0,C 180,E1 -14321.896,E2 -14321.896} C_VEL
LIN {X 0,Y 340.815,Z 298.027,A -85,B 0,C 180,E1 -14325.546,E2 -14325.546} C_VEL
LIN {X 0,Y 340.73,Z 298.04,A -85,B 0,C 180,E1 -14329.265,E2 -14329.265} C_VEL
LIN {X 0,Y 340.702,Z 298.048,A -85,B 0,C 180,E1 -14333.07,E2 -14333.07} C_VEL
LIN {X 0,Y 340.71,Z 298.042,A -85,B 0,C 180,E1 -14335.664,E2 -14335.664} C_VEL
LIN {X 0,Y 340.693,Z 298.047,A -85,B 0,C 180,E1 -14339.669,E2 -14339.669} C_VEL
LIN {X 0,Y 340.671,Z 298.045,A -85,B 0,C 180,E1 -14342.431,E2 -14342.431} C_VEL
LIN {X 0,Y 340.7,Z 298.043,A -85,B 0,C 180,E1 -14345.274,E2 -14345.274} C_VEL
LIN {X 0,Y 340.687,Z 298.044,A -85,B 0,C 180,E1 -14346.615,E2 -14346.615} C_VEL
LIN {X 0,Y 340.007,Z 298.134,A -85,B 0,C 180,E1 -14347.601,E2 -14347.601} C_VEL
LIN {X 0,Y 337.121,Z 298.488,A -85,B 0,C 180,E1 -14349.204,E2 -14349.204} C_VEL
LIN {X 0,Y 334.691,Z 298.792,A -85,B 0,C 180,E1 -14350.502,E2 -14350.502} C_VEL
LIN {X 0,Y 333.664,Z 298.919,A -85,B 0,C 180,E1 -14351.507,E2 -14351.507} C_VEL
LIN {X 0,Y 333.59,Z 298.927,A -85,B 0,C 180,E1 -14351.847,E2 -14351.847} C_VEL
LIN {X 0,Y 333.566,Z 298.931,A -85,B 0,C 180,E1 -14355.745,E2 -14355.745} C_VEL
LIN {X 0,Y 333.619,Z 298.924,A -85,B 0,C 180,E1 -14359.311,E2 -14359.311} C_VEL
LIN {X 0,Y 333.631,Z 298.925,A -85,B 0,C 180,E1 -14363.164,E2 -14363.164} C_VEL
LIN {X 0,Y 333.638,Z 298.924,A -85,B 0,C 180,E1 -14365.336,E2 -14365.336} C_VEL
LIN {X 0,Y 333.667,Z 298.919,A -85,B 0,C 180,E1 -14369.706,E2 -14369.706} C_VEL
LIN {X 0,Y 333.704,Z 298.913,A -85,B 0,C 180,E1 -14372.397,E2 -14372.397} C_VEL
LIN {X 0,Y 333.685,Z 298.918,A -85,B 0,C 180,E1 -14375.087,E2 -14375.087} C_VEL
LIN {X 0,Y 333.611,Z 298.926,A -85,B 0,C 180,E1 -14379.014,E2 -14379.014} C_VEL
LIN {X 0,Y 333.665,Z 298.918,A -85,B 0,C 180,E1 -14382.849,E2 -14382.849} C_VEL
LIN {X 0,Y 333.764,Z 298.908,A -85,B 0,C 180,E1 -14385.575,E2 -14385.575} C_VEL
LIN {X 0,Y 333.788,Z 298.903,A -85,B 0,C 180,E1 -14389.076,E2 -14389.076} C_VEL
LIN {X 0,Y 333.958,Z 298.885,A -85,B 0,C 180,E1 -14392.745,E2 -14392.745} C_VEL
LIN {X 0,Y 333.765,Z 298.907,A -85,B 0,C 180,E1 -14395.168,E2 -14395.168} C_VEL
LIN {X 0,Y 334.088,Z 298.865,A -85,B 0,C 180,E1 -14397.588,E2 -14397.588} C_VEL
LIN {X 0,Y 334.177,Z 298.854,A -85,B 0,C 180,E1 -14399.999,E2 -14399.999} C_VEL
LIN {X 0,Y 334.057,Z 298.87,A -85,B 0,C 180,E1 -14402.411,E2 -14402.411} C_VEL
LIN {X 0,Y 333.964,Z 298.881,A -85,B 0,C 180,E1 -14406.039,E2 -14406.039} C_VEL
LIN {X 0,Y 333.802,Z 298.905,A -85,B 0,C 180,E1 -14409.696,E2 -14409.696} C_VEL
LIN {X 0,Y 333.746,Z 298.912,A -85,B 0,C 180,E1 -14413.393,E2 -14413.393} C_VEL
LIN {X 0,Y 333.695,Z 298.915,A -85,B 0,C 180,E1 -14417.148,E2 -14417.148} C_VEL
LIN {X 0,Y 333.681,Z 298.919,A -85,B 0,C 180,E1 -14419.693,E2 -14419.693} C_VEL
LIN {X 0,Y 333.628,Z 298.923,A -85,B 0,C 180,E1 -14423.593,E2 -14423.593} C_VEL
LIN {X 0,Y 333.686,Z 298.92,A -85,B 0,C 180,E1 -14426.25,E2 -14426.25} C_VEL
LIN {X 0,Y 333.637,Z 298.924,A -85,B 0,C 180,E1 -14428.978,E2 -14428.978} C_VEL
LIN {X 0,Y 333.597,Z 298.929,A -85,B 0,C 180,E1 -14433.212,E2 -14433.212} C_VEL
LIN {X 0,Y 333.638,Z 298.922,A -85,B 0,C 180,E1 -14436.143,E2 -14436.143} C_VEL
LIN {X 0,Y 333.611,Z 298.931,A -85,B 0,C 180,E1 -14439.197,E2 -14439.197} C_VEL
LIN {X 0,Y 333.599,Z 298.926,A -85,B 0,C 180,E1 -14442.503,E2 -14442.503} C_VEL
LIN {X 0,Y 333.565,Z 298.933,A -85,B 0,C 180,E1 -14445.959,E2 -14445.959} C_VEL
LIN {X 0,Y 333.617,Z 298.927,A -85,B 0,C 180,E1 -14449.321,E2 -14449.321} C_VEL
LIN {X 0,Y 333.636,Z 298.922,A -85,B 0,C 180,E1 -14453.173,E2 -14453.173} C_VEL
LIN {X 0,Y 333.615,Z 298.925,A -85,B 0,C 180,E1 -14456.796,E2 -14456.796} C_VEL
LIN {X 0,Y 333.709,Z 299.111,A -85,B 0,C 180,E1 -14458.399,E2 -14458.399} C_VEL
LIN {X 0,Y 336.631,Z 312.325,A -85,B 0,C 180,E1 -14461.54,E2 -14461.54} C_VEL
LIN {X 0,Y 338.994,Z 323.946,A -85,B 0,C 180,E1 -14464.197,E2 -14464.197} C_VEL
LIN {X 0,Y 337.346,Z 339.163,A -85,B 0,C 180,E1 -14467.336,E2 -14467.336} C_VEL
LIN {X 0,Y 336.735,Z 344.269,A -85,B 0,C 180,E1 -14468.382,E2 -14468.382} C_VEL
LIN {X 0,Y 339.737,Z 373.272,A -85,B 0,C 180,E1 -14469.272,E2 -14469.272} C_VEL
LIN {X 0,Y 338.094,Z 447.932,A -85,B 0,C 180,E1 -14471.13,E2 -14471.13} C_VEL
LIN {X 0,Y 337.7,Z 457.555,A -85,B 0,C 180,E1 -14471.5,E2 -14471.5} C_VEL
LIN {X 0,Y 337.141,Z 467.334,A -85,B 0,C 180,E1 -14472.019,E2 -14472.019} C_VEL
LIN {X 0,Y 336.498,Z 477.035,A -85,B 0,C 180,E1 -14472.69,E2 -14472.69} C_VEL
LIN {X 0,Y 335.862,Z 485.764,A -85,B 0,C 180,E1 -14473.439,E2 -14473.439} C_VEL
LIN {X 0,Y 335.101,Z 495.515,A -85,B 0,C 180,E1 -14474.474,E2 -14474.474} C_VEL
LIN {X 0,Y 334.401,Z 503.913,A -85,B 0,C 180,E1 -14475.552,E2 -14475.552} C_VEL
LIN {X 0,Y 333.836,Z 510.95,A -85,B 0,C 180,E1 -14476.614,E2 -14476.614} C_VEL
LIN {X 0,Y 333.233,Z 519.267,A -85,B 0,C 180,E1 -14478.137,E2 -14478.137} C_VEL
LIN {X 0,Y 332.733,Z 526.122,A -85,B 0,C 180,E1 -14479.661,E2 -14479.661} C_VEL
LIN {X 0,Y 332.464,Z 530.81,A -85,B 0,C 180,E1 -14480.881,E2 -14480.881} C_VEL
LIN {X 0,Y 332.255,Z 536.445,A -85,B 0,C 180,E1 -14482.712,E2 -14482.712} C_VEL
LIN {X 0,Y 332.114,Z 540.598,A -85,B 0,C 180,E1 -14484.439,E2 -14484.439} C_VEL
LIN {X 0,Y 332.145,Z 543.121,A -85,B 0,C 180,E1 -14485.756,E2 -14485.756} C_VEL
LIN {X 0,Y 332.153,Z 545.586,A -85,B 0,C 180,E1 -14487.577,E2 -14487.577} C_VEL
LIN {X 0,Y 332.279,Z 546.57,A -85,B 0,C 180,E1 -14488.791,E2 -14488.791} C_VEL
LIN {X 0,Y 332.266,Z 547.192,A -85,B 0,C 180,E1 -14490.002,E2 -14490.002} C_VEL
LIN {X 0,Y 332.158,Z 547.43,A -85,B 0,C 180,E1 -14491.215,E2 -14491.215} C_VEL
LIN {X 0,Y 332.04,Z 546.385,A -85,B 0,C 180,E1 -14493.643,E2 -14493.643} C_VEL
LIN {X 0,Y 332.008,Z 545.298,A -85,B 0,C 180,E1 -14494.859,E2 -14494.859} C_VEL
LIN {X 0,Y 332.114,Z 542.754,A -85,B 0,C 180,E1 -14496.685,E2 -14496.685} C_VEL
LIN {X 0,Y 332.355,Z 539.162,A -85,B 0,C 180,E1 -14498.514,E2 -14498.514} C_VEL
LIN {X 0,Y 332.835,Z 534.432,A -85,B 0,C 180,E1 -14500.341,E2 -14500.341} C_VEL
LIN {X 0,Y 333.57,Z 528.389,A -85,B 0,C 180,E1 -14502.164,E2 -14502.164} C_VEL
LIN {X 0,Y 334.71,Z 520.802,A -85,B 0,C 180,E1 -14503.974,E2 -14503.974} C_VEL
LIN {X 0,Y 335.702,Z 513.313,A -85,B 0,C 180,E1 -14505.451,E2 -14505.451} C_VEL
LIN {X 0,Y 336.792,Z 505.877,A -85,B 0,C 180,E1 -14506.675,E2 -14506.675} C_VEL
LIN {X 0,Y 338.068,Z 497.226,A -85,B 0,C 180,E1 -14507.857,E2 -14507.857} C_VEL
LIN {X 0,Y 339.329,Z 488.138,A -85,B 0,C 180,E1 -14508.882,E2 -14508.882} C_VEL
LIN {X 0,Y 340.521,Z 478.684,A -85,B 0,C 180,E1 -14509.753,E2 -14509.753} C_VEL
LIN {X 0,Y 341.584,Z 468.934,A -85,B 0,C 180,E1 -14510.474,E2 -14510.474} C_VEL
LIN {X 0,Y 342.412,Z 459.006,A -85,B 0,C 180,E1 -14511.051,E2 -14511.051} C_VEL
LIN {X 0,Y 343.208,Z 447.887,A -85,B 0,C 180,E1 -14511.511,E2 -14511.511} C_VEL
LIN {X 0,Y 344.151,Z 422.734,A -85,B 0,C 180,E1 -14512.197,E2 -14512.197} C_VEL
LIN {X 0,Y 345.956,Z 373.205,A -85,B 0,C 180,E1 -14513.502,E2 -14513.502} C_VEL
LIN {X 0,Y 343.513,Z 355.069,A -85,B 0,C 180,E1 -14514.31,E2 -14514.31} C_VEL
LIN {X 0,Y 341.18,Z 342.834,A -85,B 0,C 180,E1 -14514.994,E2 -14514.994} C_VEL
LIN {X 0,Y 342.586,Z 332.244,A -85,B 0,C 180,E1 -14517.046,E2 -14517.046} C_VEL
LIN {X 0,Y 341.547,Z 325.682,A -85,B 0,C 180,E1 -14518.572,E2 -14518.572} C_VEL
LIN {X 0,Y 338.967,Z 315.314,A -85,B 0,C 180,E1 -14521.22,E2 -14521.22} C_VEL
LIN {X 0,Y 335.921,Z 305.373,A -85,B 0,C 180,E1 -14524.051,E2 -14524.051} C_VEL
LIN {X 0,Y 333.669,Z 298.925,A -85,B 0,C 180,E1 -14526.139,E2 -14526.139} C_VEL
LIN {X 0,Y 333.638,Z 298.932,A -85,B 0,C 180,E1 -14529.192,E2 -14529.192} C_VEL
LIN {X 0,Y 333.623,Z 298.932,A -85,B 0,C 180,E1 -14532.499,E2 -14532.499} C_VEL
LIN {X 0,Y 333.585,Z 298.931,A -85,B 0,C 180,E1 -14535.954,E2 -14535.954} C_VEL
LIN {X 0,Y 333.643,Z 298.926,A -85,B 0,C 180,E1 -14539.313,E2 -14539.313} C_VEL
LIN {X 0,Y 333.64,Z 298.919,A -85,B 0,C 180,E1 -14542.348,E2 -14542.348} C_VEL
LIN {X 0,Y 333.659,Z 298.915,A -85,B 0,C 180,E1 -14545.34,E2 -14545.34} C_VEL
LIN {X 0,Y 333.688,Z 298.909,A -85,B 0,C 180,E1 -14549.71,E2 -14549.71} C_VEL
LIN {X 0,Y 333.726,Z 298.908,A -85,B 0,C 180,E1 -14552.4,E2 -14552.4} C_VEL
LIN {X 0,Y 333.715,Z 298.916,A -85,B 0,C 180,E1 -14555.09,E2 -14555.09} C_VEL
LIN {X 0,Y 333.691,Z 298.918,A -85,B 0,C 180,E1 -14559.021,E2 -14559.021} C_VEL
LIN {X 0,Y 333.776,Z 298.91,A -85,B 0,C 180,E1 -14561.589,E2 -14561.589} C_VEL
LIN {X 0,Y 333.79,Z 298.907,A -85,B 0,C 180,E1 -14565.577,E2 -14565.577} C_VEL
LIN {X 0,Y 333.802,Z 299.045,A -85,B 0,C 180,E1 -14568.27,E2 -14568.27} C_VEL
LIN {X 0,Y 337.862,Z 310.405,A -85,B 0,C 180,E1 -14571.628,E2 -14571.628} C_VEL
LIN {X 0,Y 339.802,Z 317.211,A -85,B 0,C 180,E1 -14573.409,E2 -14573.409} C_VEL
LIN {X 0,Y 341.388,Z 325.088,A -85,B 0,C 180,E1 -14575.277,E2 -14575.277} C_VEL
LIN {X 0,Y 340.117,Z 338.863,A -85,B 0,C 180,E1 -14577.891,E2 -14577.891} C_VEL
LIN {X 0,Y 343.859,Z 357.418,A -85,B 0,C 180,E1 -14578.976,E2 -14578.976} C_VEL
LIN {X 0,Y 345.623,Z 369.021,A -85,B 0,C 180,E1 -14579.563,E2 -14579.563} C_VEL
LIN {X 0,Y 342.892,Z 426.972,A -85,B 0,C 180,E1 -14581.359,E2 -14581.359} C_VEL
LIN {X 0,Y 342.125,Z 438.756,A -85,B 0,C 180,E1 -14581.914,E2 -14581.914} C_VEL
LIN {X 0,Y 341.18,Z 449.676,A -85,B 0,C 180,E1 -14582.657,E2 -14582.657} C_VEL
LIN {X 0,Y 340.184,Z 459.716,A -85,B 0,C 180,E1 -14583.554,E2 -14583.554} C_VEL
LIN {X 0,Y 339.215,Z 467.893,A -85,B 0,C 180,E1 -14584.457,E2 -14584.457} C_VEL
LIN {X 0,Y 338.141,Z 475.82,A -85,B 0,C 180,E1 -14585.518,E2 -14585.518} C_VEL
LIN {X 0,Y 337.197,Z 482.412,A -85,B 0,C 180,E1 -14586.583,E2 -14586.583} C_VEL
LIN {X 0,Y 336.249,Z 488.738,A -85,B 0,C 180,E1 -14587.809,E2 -14587.809} C_VEL
LIN {X 0,Y 335.413,Z 494.023,A -85,B 0,C 180,E1 -14589.042,E2 -14589.042} C_VEL
LIN {X 0,Y 334.668,Z 498.441,A -85,B 0,C 180,E1 -14590.283,E2 -14590.283} C_VEL
LIN {X 0,Y 334.015,Z 502.109,A -85,B 0,C 180,E1 -14591.531,E2 -14591.531} C_VEL
LIN {X 0,Y 333.29,Z 506.308,A -85,B 0,C 180,E1 -14593.413,E2 -14593.413} C_VEL
LIN {X 0,Y 332.887,Z 508.337,A -85,B 0,C 180,E1 -14594.676,E2 -14594.676} C_VEL
LIN {X 0,Y 332.559,Z 509.803,A -85,B 0,C 180,E1 -14595.947,E2 -14595.947} C_VEL
LIN {X 0,Y 332.303,Z 510.705,A -85,B 0,C 180,E1 -14597.224,E2 -14597.224} C_VEL
LIN {X 0,Y 332.144,Z 510.954,A -85,B 0,C 180,E1 -14598.506,E2 -14598.506} C_VEL
LIN {X 0,Y 332.024,Z 510.612,A -85,B 0,C 180,E1 -14599.797,E2 -14599.797} C_VEL
LIN {X 0,Y 332.033,Z 509.451,A -85,B 0,C 180,E1 -14601.365,E2 -14601.365} C_VEL
LIN {X 0,Y 332.162,Z 507.239,A -85,B 0,C 180,E1 -14603.044,E2 -14603.044} C_VEL
LIN {X 0,Y 332.427,Z 503.298,A -85,B 0,C 180,E1 -14605.014,E2 -14605.014} C_VEL
LIN {X 0,Y 332.713,Z 498.702,A -85,B 0,C 180,E1 -14606.644,E2 -14606.644} C_VEL
LIN {X 0,Y 333.062,Z 493.895,A -85,B 0,C 180,E1 -14608.003,E2 -14608.003} C_VEL
LIN {X 0,Y 333.43,Z 488.091,A -85,B 0,C 180,E1 -14609.345,E2 -14609.345} C_VEL
LIN {X 0,Y 333.971,Z 481.012,A -85,B 0,C 180,E1 -14610.685,E2 -14610.685} C_VEL
LIN {X 0,Y 334.549,Z 473.497,A -85,B 0,C 180,E1 -14611.858,E2 -14611.858} C_VEL
LIN {X 0,Y 335.056,Z 465.63,A -85,B 0,C 180,E1 -14612.878,E2 -14612.878} C_VEL
LIN {X 0,Y 335.695,Z 456.173,A -85,B 0,C 180,E1 -14613.878,E2 -14613.878} C_VEL
LIN {X 0,Y 336.414,Z 443.679,A -85,B 0,C 180,E1 -14614.883,E2 -14614.883} C_VEL
LIN {X 0,Y 336.784,Z 433.456,A -85,B 0,C 180,E1 -14615.484,E2 -14615.484} C_VEL
LIN {X 0,Y 337.148,Z 423.647,A -85,B 0,C 180,E1 -14615.894,E2 -14615.894} C_VEL
LIN {X 0,Y 338.527,Z 365.498,A -85,B 0,C 180,E1 -14617.517,E2 -14617.517} C_VEL
LIN {X 0,Y 335.273,Z 339.772,A -85,B 0,C 180,E1 -14618.405,E2 -14618.405} C_VEL
LIN {X 0,Y 336.516,Z 323.758,A -85,B 0,C 180,E1 -14622.341,E2 -14622.341} C_VEL
LIN {X 0,Y 337.033,Z 316.342,A -85,B 0,C 180,E1 -14624.201,E2 -14624.201} C_VEL
LIN {X 0,Y 334.932,Z 305.122,A -85,B 0,C 180,E1 -14627.259,E2 -14627.259} C_VEL
LIN {X 0,Y 333.681,Z 298.922,A -85,B 0,C 180,E1 -14629.04,E2 -14629.04} C_VEL
LIN {X 0,Y 333.659,Z 298.921,A -85,B 0,C 180,E1 -14633.17,E2 -14633.17} C_VEL
LIN {X 0,Y 333.672,Z 298.92,A -85,B 0,C 180,E1 -14635.342,E2 -14635.342} C_VEL
LIN {X 0,Y 333.628,Z 298.926,A -85,B 0,C 180,E1 -14638.222,E2 -14638.222} C_VEL
LIN {X 0,Y 333.63,Z 298.922,A -85,B 0,C 180,E1 -14641.021,E2 -14641.021} C_VEL
LIN {X 0,Y 333.658,Z 298.92,A -85,B 0,C 180,E1 -14644.923,E2 -14644.923} C_VEL
LIN {X 0,Y 333.659,Z 298.921,A -85,B 0,C 180,E1 -14649.017,E2 -14649.017} C_VEL
LIN {X 0,Y 333.745,Z 298.908,A -85,B 0,C 180,E1 -14651.586,E2 -14651.586} C_VEL
LIN {X 0,Y 333.814,Z 298.9,A -85,B 0,C 180,E1 -14655.576,E2 -14655.576} C_VEL
LIN {X 0,Y 333.821,Z 298.905,A -85,B 0,C 180,E1 -14659.076,E2 -14659.076} C_VEL
LIN {X 0,Y 333.96,Z 298.883,A -85,B 0,C 180,E1 -14662.744,E2 -14662.744} C_VEL
LIN {X 0,Y 333.777,Z 298.908,A -85,B 0,C 180,E1 -14665.167,E2 -14665.167} C_VEL
LIN {X 0,Y 334.061,Z 298.876,A -85,B 0,C 180,E1 -14667.586,E2 -14667.586} C_VEL
LIN {X 0,Y 334.061,Z 298.87,A -85,B 0,C 180,E1 -14671.203,E2 -14671.203} C_VEL
LIN {X 0,Y 334.061,Z 298.87,A -85,B 0,C 180,E1 -14672.409,E2 -14672.409} C_VEL
LIN {X 0,Y 333.987,Z 298.884,A -85,B 0,C 180,E1 -14676.036,E2 -14676.036} C_VEL
LIN {X 0,Y 333.914,Z 298.891,A -85,B 0,C 180,E1 -14678.469,E2 -14678.469} C_VEL
LIN {X 0,Y 333.789,Z 298.906,A -85,B 0,C 180,E1 -14682.151,E2 -14682.151} C_VEL
LIN {X 0,Y 333.807,Z 298.907,A -85,B 0,C 180,E1 -14684.63,E2 -14684.63} C_VEL
LIN {X 0,Y 333.72,Z 298.916,A -85,B 0,C 180,E1 -14688.613,E2 -14688.613} C_VEL
LIN {X 0,Y 333.645,Z 298.921,A -85,B 0,C 180,E1 -14692.276,E2 -14692.276} C_VEL
LIN {X 0,Y 333.68,Z 298.922,A -85,B 0,C 180,E1 -14695.085,E2 -14695.085} C_VEL
LIN {X 0,Y 333.641,Z 298.923,A -85,B 0,C 180,E1 -14698.973,E2 -14698.973} C_VEL
LIN {X 0,Y 333.629,Z 298.922,A -85,B 0,C 180,E1 -14702.582,E2 -14702.582} C_VEL
LIN {X 0,Y 333.658,Z 298.922,A -85,B 0,C 180,E1 -14706.134,E2 -14706.134} C_VEL
LIN {X 0,Y 333.625,Z 298.923,A -85,B 0,C 180,E1 -14709.187,E2 -14709.187} C_VEL
LIN {X 0,Y 333.59,Z 298.927,A -85,B 0,C 180,E1 -14711.847,E2 -14711.847} C_VEL
LIN {X 0,Y 332.95,Z 299.011,A -85,B 0,C 180,E1 -14712.855,E2 -14712.855} C_VEL
LIN {X 0,Y 330.117,Z 299.367,A -85,B 0,C 180,E1 -14714.495,E2 -14714.495} C_VEL
LIN {X 0,Y 327.691,Z 299.667,A -85,B 0,C 180,E1 -14715.823,E2 -14715.823} C_VEL
LIN {X 0,Y 326.634,Z 299.797,A -85,B 0,C 180,E1 -14716.851,E2 -14716.851} C_VEL
LIN {X 0,Y 326.54,Z 299.806,A -85,B 0,C 180,E1 -14717.199,E2 -14717.199} C_VEL
LIN {X 0,Y 326.581,Z 299.806,A -85,B 0,C 180,E1 -14720.768,E2 -14720.768} C_VEL
LIN {X 0,Y 326.577,Z 299.804,A -85,B 0,C 180,E1 -14724.475,E2 -14724.475} C_VEL
LIN {X 0,Y 326.57,Z 299.804,A -85,B 0,C 180,E1 -14727.451,E2 -14727.451} C_VEL
LIN {X 0,Y 326.624,Z 299.795,A -85,B 0,C 180,E1 -14730.337,E2 -14730.337} C_VEL
LIN {X 0,Y 326.651,Z 299.792,A -85,B 0,C 180,E1 -14734.512,E2 -14734.512} C_VEL
LIN {X 0,Y 326.568,Z 299.802,A -85,B 0,C 180,E1 -14738.539,E2 -14738.539} C_VEL
LIN {X 0,Y 326.628,Z 299.796,A -85,B 0,C 180,E1 -14741.191,E2 -14741.191} C_VEL
LIN {X 0,Y 326.719,Z 299.784,A -85,B 0,C 180,E1 -14745.432,E2 -14745.432} C_VEL
LIN {X 0,Y 326.724,Z 299.784,A -85,B 0,C 180,E1 -14748.837,E2 -14748.837} C_VEL
LIN {X 0,Y 326.908,Z 299.765,A -85,B 0,C 180,E1 -14752.588,E2 -14752.588} C_VEL
LIN {X 0,Y 326.731,Z 299.784,A -85,B 0,C 180,E1 -14755.063,E2 -14755.063} C_VEL
LIN {X 0,Y 327.026,Z 299.745,A -85,B 0,C 180,E1 -14757.536,E2 -14757.536} C_VEL
LIN {X 0,Y 327.129,Z 299.732,A -85,B 0,C 180,E1 -14759.999,E2 -14759.999} C_VEL
LIN {X 0,Y 326.998,Z 299.75,A -85,B 0,C 180,E1 -14762.463,E2 -14762.463} C_VEL
LIN {X 0,Y 326.939,Z 299.756,A -85,B 0,C 180,E1 -14766.17,E2 -14766.17} C_VEL
LIN {X 0,Y 326.758,Z 299.781,A -85,B 0,C 180,E1 -14769.907,E2 -14769.907} C_VEL
LIN {X 0,Y 326.71,Z 299.791,A -85,B 0,C 180,E1 -14773.687,E2 -14773.687} C_VEL
LIN {X 0,Y 326.645,Z 299.795,A -85,B 0,C 180,E1 -14777.53,E2 -14777.53} C_VEL
LIN {X 0,Y 326.609,Z 299.803,A -85,B 0,C 180,E1 -14780.138,E2 -14780.138} C_VEL
LIN {X 0,Y 326.607,Z 299.802,A -85,B 0,C 180,E1 -14784.132,E2 -14784.132} C_VEL
LIN {X 0,Y 326.633,Z 299.796,A -85,B 0,C 180,E1 -14786.861,E2 -14786.861} C_VEL
LIN {X 0,Y 326.572,Z 299.808,A -85,B 0,C 180,E1 -14790.606,E2 -14790.606} C_VEL
LIN {X 0,Y 326.568,Z 299.802,A -85,B 0,C 180,E1 -14794.023,E2 -14794.023} C_VEL
LIN {X 0,Y 326.59,Z 299.804,A -85,B 0,C 180,E1 -14797.242,E2 -14797.242} C_VEL
LIN {X 0,Y 326.544,Z 299.811,A -85,B 0,C 180,E1 -14801.135,E2 -14801.135} C_VEL
LIN {X 0,Y 326.495,Z 299.812,A -85,B 0,C 180,E1 -14804.746,E2 -14804.746} C_VEL
LIN {X 0,Y 326.547,Z 299.806,A -85,B 0,C 180,E1 -14808.158,E2 -14808.158} C_VEL
LIN {X 0,Y 326.56,Z 299.805,A -85,B 0,C 180,E1 -14811.39,E2 -14811.39} C_VEL
LIN {X 0,Y 326.594,Z 299.799,A -85,B 0,C 180,E1 -14814.857,E2 -14814.857} C_VEL
LIN {X 0,Y 326.613,Z 299.804,A -85,B 0,C 180,E1 -14818.009,E2 -14818.009} C_VEL
LIN {X 0,Y 329.763,Z 314.023,A -85,B 0,C 180,E1 -14821.47,E2 -14821.47} C_VEL
LIN {X 0,Y 331.962,Z 324.62,A -85,B 0,C 180,E1 -14823.946,E2 -14823.946} C_VEL
LIN {X 0,Y 331.624,Z 329.217,A -85,B 0,C 180,E1 -14824.927,E2 -14824.927} C_VEL
LIN {X 0,Y 329.825,Z 344.385,A -85,B 0,C 180,E1 -14828.092,E2 -14828.092} C_VEL
LIN {X 0,Y 332.834,Z 373.942,A -85,B 0,C 180,E1 -14829.01,E2 -14829.01} C_VEL
LIN {X 0,Y 331.155,Z 447.371,A -85,B 0,C 180,E1 -14830.88,E2 -14830.88} C_VEL
LIN {X 0,Y 330.758,Z 457.068,A -85,B 0,C 180,E1 -14831.258,E2 -14831.258} C_VEL
LIN {X 0,Y 330.186,Z 466.876,A -85,B 0,C 180,E1 -14831.787,E2 -14831.787} C_VEL
LIN {X 0,Y 329.52,Z 476.595,A -85,B 0,C 180,E1 -14832.471,E2 -14832.471} C_VEL
LIN {X 0,Y 328.877,Z 485.344,A -85,B 0,C 180,E1 -14833.237,E2 -14833.237} C_VEL
LIN {X 0,Y 328.156,Z 494.245,A -85,B 0,C 180,E1 -14834.186,E2 -14834.186} C_VEL
LIN {X 0,Y 327.356,Z 503.511,A -85,B 0,C 180,E1 -14835.393,E2 -14835.393} C_VEL
LIN {X 0,Y 326.7,Z 511.424,A -85,B 0,C 180,E1 -14836.633,E2 -14836.633} C_VEL
LIN {X 0,Y 326.235,Z 518.159,A -85,B 0,C 180,E1 -14837.879,E2 -14837.879} C_VEL
LIN {X 0,Y 325.694,Z 525.14,A -85,B 0,C 180,E1 -14839.435,E2 -14839.435} C_VEL
LIN {X 0,Y 325.395,Z 529.907,A -85,B 0,C 180,E1 -14840.681,E2 -14840.681} C_VEL
LIN {X 0,Y 325.183,Z 535.673,A -85,B 0,C 180,E1 -14842.552,E2 -14842.552} C_VEL
LIN {X 0,Y 325.029,Z 540.228,A -85,B 0,C 180,E1 -14844.484,E2 -14844.484} C_VEL
LIN {X 0,Y 325.031,Z 543.377,A -85,B 0,C 180,E1 -14846.284,E2 -14846.284} C_VEL
LIN {X 0,Y 325.063,Z 544.996,A -85,B 0,C 180,E1 -14847.524,E2 -14847.524} C_VEL
LIN {X 0,Y 325.199,Z 546.042,A -85,B 0,C 180,E1 -14848.764,E2 -14848.764} C_VEL
LIN {X 0,Y 325.206,Z 546.739,A -85,B 0,C 180,E1 -14850.003,E2 -14850.003} C_VEL
LIN {X 0,Y 325.065,Z 546.981,A -85,B 0,C 180,E1 -14851.241,E2 -14851.241} C_VEL
LIN {X 0,Y 324.962,Z 546.076,A -85,B 0,C 180,E1 -14853.722,E2 -14853.722} C_VEL
LIN {X 0,Y 324.953,Z 543.956,A -85,B 0,C 180,E1 -14855.81,E2 -14855.81} C_VEL
LIN {X 0,Y 325.193,Z 540.216,A -85,B 0,C 180,E1 -14858.077,E2 -14858.077} C_VEL
LIN {X 0,Y 325.621,Z 535.948,A -85,B 0,C 180,E1 -14859.944,E2 -14859.944} C_VEL
LIN {X 0,Y 326.037,Z 532.473,A -85,B 0,C 180,E1 -14861.188,E2 -14861.188} C_VEL
LIN {X 0,Y 326.825,Z 527.287,A -85,B 0,C 180,E1 -14862.735,E2 -14862.735} C_VEL
LIN {X 0,Y 327.813,Z 521.026,A -85,B 0,C 180,E1 -14864.274,E2 -14864.274} C_VEL
LIN {X 0,Y 328.782,Z 514.194,A -85,B 0,C 180,E1 -14865.683,E2 -14865.683} C_VEL
LIN {X 0,Y 330.195,Z 505.307,A -85,B 0,C 180,E1 -14867.178,E2 -14867.178} C_VEL
LIN {X 0,Y 331.503,Z 496.613,A -85,B 0,C 180,E1 -14868.383,E2 -14868.383} C_VEL
LIN {X 0,Y 332.871,Z 487.498,A -85,B 0,C 180,E1 -14869.423,E2 -14869.423} C_VEL
LIN {X 0,Y 334.127,Z 478.06,A -85,B 0,C 180,E1 -14870.308,E2 -14870.308} C_VEL
LIN {X 0,Y 335.221,Z 468.34,A -85,B 0,C 180,E1 -14871.041,E2 -14871.041} C_VEL
LIN {X 0,Y 336.14,Z 458.434,A -85,B 0,C 180,E1 -14871.624,E2 -14871.624} C_VEL
LIN {X 0,Y 336.972,Z 447.324,A -85,B 0,C 180,E1 -14872.09,E2 -14872.09} C_VEL
LIN {X 0,Y 338.03,Z 420.865,A -85,B 0,C 180,E1 -14872.823,E2 -14872.823} C_VEL
LIN {X 0,Y 339.825,Z 374.145,A -85,B 0,C 180,E1 -14874.087,E2 -14874.087} C_VEL
LIN {X 0,Y 337.593,Z 356.879,A -85,B 0,C 180,E1 -14874.895,E2 -14874.895} C_VEL
LIN {X 0,Y 334.906,Z 342.855,A -85,B 0,C 180,E1 -14875.69,E2 -14875.69} C_VEL
LIN {X 0,Y 336.097,Z 334.297,A -85,B 0,C 180,E1 -14877.389,E2 -14877.389} C_VEL
LIN {X 0,Y 334.607,Z 325.863,A -85,B 0,C 180,E1 -14879.456,E2 -14879.456} C_VEL
LIN {X 0,Y 331.841,Z 315.288,A -85,B 0,C 180,E1 -14882.326,E2 -14882.326} C_VEL
LIN {X 0,Y 329.297,Z 307.335,A -85,B 0,C 180,E1 -14884.748,E2 -14884.748} C_VEL
LIN {X 0,Y 326.6,Z 299.807,A -85,B 0,C 180,E1 -14887.314,E2 -14887.314} C_VEL
LIN {X 0,Y 326.569,Z 299.81,A -85,B 0,C 180,E1 -14891.13,E2 -14891.13} C_VEL
LIN {X 0,Y 326.517,Z 299.815,A -85,B 0,C 180,E1 -14894.742,E2 -14894.742} C_VEL
LIN {X 0,Y 326.569,Z 299.804,A -85,B 0,C 180,E1 -14898.154,E2 -14898.154} C_VEL
LIN {X 0,Y 326.627,Z 299.799,A -85,B 0,C 180,E1 -14901.393,E2 -14901.393} C_VEL
LIN {X 0,Y 326.605,Z 299.792,A -85,B 0,C 180,E1 -14904.851,E2 -14904.851} C_VEL
LIN {X 0,Y 326.593,Z 299.792,A -85,B 0,C 180,E1 -14907.455,E2 -14907.455} C_VEL
LIN {X 0,Y 326.645,Z 299.79,A -85,B 0,C 180,E1 -14910.34,E2 -14910.34} C_VEL
LIN {X 0,Y 326.676,Z 299.788,A -85,B 0,C 180,E1 -14914.516,E2 -14914.516} C_VEL
LIN {X 0,Y 326.644,Z 299.794,A -85,B 0,C 180,E1 -14918.546,E2 -14918.546} C_VEL
LIN {X 0,Y 326.728,Z 299.786,A -85,B 0,C 180,E1 -14921.177,E2 -14921.177} C_VEL
LIN {X 0,Y 326.744,Z 299.786,A -85,B 0,C 180,E1 -14925.434,E2 -14925.434} C_VEL
LIN {X 0,Y 326.751,Z 299.881,A -85,B 0,C 180,E1 -14927.067,E2 -14927.067} C_VEL
LIN {X 0,Y 330.575,Z 310.352,A -85,B 0,C 180,E1 -14930.419,E2 -14930.419} C_VEL
LIN {X 0,Y 333.153,Z 318.584,A -85,B 0,C 180,E1 -14932.729,E2 -14932.729} C_VEL
LIN {X 0,Y 334.993,Z 327.297,A -85,B 0,C 180,E1 -14934.897,E2 -14934.897} C_VEL
LIN {X 0,Y 333.741,Z 338.631,A -85,B 0,C 180,E1 -14937.134,E2 -14937.134} C_VEL
LIN {X 0,Y 337.596,Z 357.185,A -85,B 0,C 180,E1 -14938.288,E2 -14938.288} C_VEL
LIN {X 0,Y 339.503,Z 370.461,A -85,B 0,C 180,E1 -14938.997,E2 -14938.997} C_VEL
LIN {X 0,Y 336.662,Z 427.092,A -85,B 0,C 180,E1 -14940.789,E2 -14940.789} C_VEL
LIN {X 0,Y 335.845,Z 438.874,A -85,B 0,C 180,E1 -14941.35,E2 -14941.35} C_VEL
LIN {X 0,Y 334.857,Z 449.87,A -85,B 0,C 180,E1 -14942.106,E2 -14942.106} C_VEL
LIN {X 0,Y 333.767,Z 459.898,A -85,B 0,C 180,E1 -14943.018,E2 -14943.018} C_VEL
LIN {X 0,Y 332.744,Z 468.055,A -85,B 0,C 180,E1 -14943.937,E2 -14943.937} C_VEL
LIN {X 0,Y 331.58,Z 476.141,A -85,B 0,C 180,E1 -14945.043,E2 -14945.043} C_VEL
LIN {X 0,Y 330.587,Z 482.605,A -85,B 0,C 180,E1 -14946.102,E2 -14946.102} C_VEL
LIN {X 0,Y 329.558,Z 488.984,A -85,B 0,C 180,E1 -14947.352,E2 -14947.352} C_VEL
LIN {X 0,Y 328.653,Z 494.308,A -85,B 0,C 180,E1 -14948.61,E2 -14948.61} C_VEL
LIN {X 0,Y 327.856,Z 498.756,A -85,B 0,C 180,E1 -14949.875,E2 -14949.875} C_VEL
LIN {X 0,Y 327.167,Z 502.449,A -85,B 0,C 180,E1 -14951.148,E2 -14951.148} C_VEL
LIN {X 0,Y 326.579,Z 505.474,A -85,B 0,C 180,E1 -14952.428,E2 -14952.428} C_VEL
LIN {X 0,Y 326.017,Z 508.33,A -85,B 0,C 180,E1 -14954.066,E2 -14954.066} C_VEL
LIN {X 0,Y 325.731,Z 509.529,A -85,B 0,C 180,E1 -14955.006,E2 -14955.006} C_VEL
LIN {X 0,Y 325.388,Z 510.665,A -85,B 0,C 180,E1 -14956.308,E2 -14956.308} C_VEL
LIN {X 0,Y 325.119,Z 511.323,A -85,B 0,C 180,E1 -14957.995,E2 -14957.995} C_VEL
LIN {X 0,Y 325.024,Z 511.304,A -85,B 0,C 180,E1 -14958.927,E2 -14958.927} C_VEL
LIN {X 0,Y 324.925,Z 510.771,A -85,B 0,C 180,E1 -14960.248,E2 -14960.248} C_VEL
LIN {X 0,Y 324.951,Z 509.57,A -85,B 0,C 180,E1 -14961.573,E2 -14961.573} C_VEL
LIN {X 0,Y 325.162,Z 506.645,A -85,B 0,C 180,E1 -14963.57,E2 -14963.57} C_VEL
LIN {X 0,Y 325.308,Z 503.976,A -85,B 0,C 180,E1 -14964.861,E2 -14964.861} C_VEL
LIN {X 0,Y 325.616,Z 499.21,A -85,B 0,C 180,E1 -14966.607,E2 -14966.607} C_VEL
LIN {X 0,Y 326.023,Z 493.158,A -85,B 0,C 180,E1 -14968.311,E2 -14968.311} C_VEL
LIN {X 0,Y 326.46,Z 487.143,A -85,B 0,C 180,E1 -14969.68,E2 -14969.68} C_VEL
LIN {X 0,Y 326.92,Z 481.173,A -85,B 0,C 180,E1 -14970.815,E2 -14970.815} C_VEL
LIN {X 0,Y 327.555,Z 473.191,A -85,B 0,C 180,E1 -14972.076,E2 -14972.076} C_VEL
LIN {X 0,Y 328.173,Z 463.839,A -85,B 0,C 180,E1 -14973.284,E2 -14973.284} C_VEL
LIN {X 0,Y 328.877,Z 452.688,A -85,B 0,C 180,E1 -14974.4,E2 -14974.4} C_VEL
LIN {X 0,Y 329.444,Z 442.648,A -85,B 0,C 180,E1 -14975.17,E2 -14975.17} C_VEL
LIN {X 0,Y 329.897,Z 432.615,A -85,B 0,C 180,E1 -14975.753,E2 -14975.753} C_VEL
LIN {X 0,Y 330.231,Z 421.481,A -85,B 0,C 180,E1 -14976.207,E2 -14976.207} C_VEL
LIN {X 0,Y 331.615,Z 366.107,A -85,B 0,C 180,E1 -14977.776,E2 -14977.776} C_VEL
LIN {X 0,Y 328.295,Z 339.763,A -85,B 0,C 180,E1 -14978.718,E2 -14978.718} C_VEL
LIN {X 0,Y 329.583,Z 324.08,A -85,B 0,C 180,E1 -14982.643,E2 -14982.643} C_VEL
LIN {X 0,Y 330.073,Z 317.737,A -85,B 0,C 180,E1 -14984.265,E2 -14984.265} C_VEL
LIN {X 0,Y 327.861,Z 305.964,A -85,B 0,C 180,E1 -14987.53,E2 -14987.53} C_VEL
LIN {X 0,Y 326.623,Z 299.802,A -85,B 0,C 180,E1 -14989.339,E2 -14989.339} C_VEL
LIN {X 0,Y 326.623,Z 299.796,A -85,B 0,C 180,E1 -14992.953,E2 -14992.953} C_VEL
LIN {X 0,Y 326.606,Z 299.802,A -85,B 0,C 180,E1 -14995.981,E2 -14995.981} C_VEL
LIN {X 0,Y 326.612,Z 299.798,A -85,B 0,C 180,E1 -14999.398,E2 -14999.398} C_VEL
LIN {X 0,Y 326.597,Z 299.798,A -85,B 0,C 180,E1 -15003.135,E2 -15003.135} C_VEL
LIN {X 0,Y 326.594,Z 299.799,A -85,B 0,C 180,E1 -15007.21,E2 -15007.21} C_VEL
LIN {X 0,Y 326.676,Z 299.79,A -85,B 0,C 180,E1 -15011.193,E2 -15011.193} C_VEL
LIN {X 0,Y 326.769,Z 299.779,A -85,B 0,C 180,E1 -15015.433,E2 -15015.433} C_VEL
LIN {X 0,Y 326.762,Z 299.782,A -85,B 0,C 180,E1 -15018.837,E2 -15018.837} C_VEL
LIN {X 0,Y 326.917,Z 299.759,A -85,B 0,C 180,E1 -15022.587,E2 -15022.587} C_VEL
LIN {X 0,Y 326.747,Z 299.782,A -85,B 0,C 180,E1 -15025.062,E2 -15025.062} C_VEL
LIN {X 0,Y 327.004,Z 299.754,A -85,B 0,C 180,E1 -15027.534,E2 -15027.534} C_VEL
LIN {X 0,Y 327.031,Z 299.746,A -85,B 0,C 180,E1 -15031.229,E2 -15031.229} C_VEL
LIN {X 0,Y 326.74,Z 299.785,A -85,B 0,C 180,E1 -15033.697,E2 -15033.697} C_VEL
LIN {X 0,Y 326.942,Z 299.761,A -85,B 0,C 180,E1 -15036.167,E2 -15036.167} C_VEL
LIN {X 0,Y 326.783,Z 299.778,A -85,B 0,C 180,E1 -15039.904,E2 -15039.904} C_VEL
LIN {X 0,Y 326.758,Z 299.779,A -85,B 0,C 180,E1 -15043.681,E2 -15043.681} C_VEL
LIN {X 0,Y 326.66,Z 299.791,A -85,B 0,C 180,E1 -15047.526,E2 -15047.526} C_VEL
LIN {X 0,Y 326.609,Z 299.799,A -85,B 0,C 180,E1 -15051.452,E2 -15051.452} C_VEL
LIN {X 0,Y 326.626,Z 299.798,A -85,B 0,C 180,E1 -15055.484,E2 -15055.484} C_VEL
LIN {X 0,Y 326.603,Z 299.802,A -85,B 0,C 180,E1 -15059.659,E2 -15059.659} C_VEL
LIN {X 0,Y 326.602,Z 299.799,A -85,B 0,C 180,E1 -15062.941,E2 -15062.941} C_VEL
LIN {X 0,Y 326.595,Z 299.803,A -85,B 0,C 180,E1 -15065.515,E2 -15065.515} C_VEL
LIN {X 0,Y 326.59,Z 299.8,A -85,B 0,C 180,E1 -15069.222,E2 -15069.222} C_VEL
LIN {X 0,Y 326.551,Z 299.805,A -85,B 0,C 180,E1 -15072.966,E2 -15072.966} C_VEL
LIN {X 0,Y 326.54,Z 299.806,A -85,B 0,C 180,E1 -15077.199,E2 -15077.199} C_VEL
LIN {X 0,Y 325.859,Z 299.895,A -85,B 0,C 180,E1 -15078.228,E2 -15078.228} C_VEL
LIN {X 0,Y 323.025,Z 300.247,A -85,B 0,C 180,E1 -15079.904,E2 -15079.904} C_VEL
LIN {X 0,Y 320.63,Z 300.546,A -85,B 0,C 180,E1 -15081.261,E2 -15081.261} C_VEL
LIN {X 0,Y 319.596,Z 300.673,A -85,B 0,C 180,E1 -15082.311,E2 -15082.311} C_VEL
LIN {X 0,Y 319.508,Z 300.682,A -85,B 0,C 180,E1 -15082.667,E2 -15082.667} C_VEL
LIN {X 0,Y 319.525,Z 300.684,A -85,B 0,C 180,E1 -15085.118,E2 -15085.118} C_VEL
LIN {X 0,Y 319.535,Z 300.684,A -85,B 0,C 180,E1 -15089.054,E2 -15089.054} C_VEL
LIN {X 0,Y 319.57,Z 300.674,A -85,B 0,C 180,E1 -15092.494,E2 -15092.494} C_VEL
LIN {X 0,Y 319.563,Z 300.679,A -85,B 0,C 180,E1 -15095.3,E2 -15095.3} C_VEL
LIN {X 0,Y 319.524,Z 300.682,A -85,B 0,C 180,E1 -15098.042,E2 -15098.042} C_VEL
LIN {X 0,Y 319.563,Z 300.679,A -85,B 0,C 180,E1 -15102.067,E2 -15102.067} C_VEL
LIN {X 0,Y 319.686,Z 300.665,A -85,B 0,C 180,E1 -15106.005,E2 -15106.005} C_VEL
LIN {X 0,Y 319.707,Z 300.659,A -85,B 0,C 180,E1 -15109.871,E2 -15109.871} C_VEL
LIN {X 0,Y 319.895,Z 300.634,A -85,B 0,C 180,E1 -15113.693,E2 -15113.693} C_VEL
LIN {X 0,Y 319.967,Z 300.625,A -85,B 0,C 180,E1 -15117.482,E2 -15117.482} C_VEL
LIN {X 0,Y 320.081,Z 300.61,A -85,B 0,C 180,E1 -15119.999,E2 -15119.999} C_VEL
LIN {X 0,Y 319.942,Z 300.629,A -85,B 0,C 180,E1 -15122.517,E2 -15122.517} C_VEL
LIN {X 0,Y 319.893,Z 300.634,A -85,B 0,C 180,E1 -15126.306,E2 -15126.306} C_VEL
LIN {X 0,Y 319.705,Z 300.658,A -85,B 0,C 180,E1 -15130.128,E2 -15130.128} C_VEL
LIN {X 0,Y 319.685,Z 300.66,A -85,B 0,C 180,E1 -15134.724,E2 -15134.724} C_VEL
LIN {X 0,Y 319.646,Z 300.664,A -85,B 0,C 180,E1 -15139.039,E2 -15139.039} C_VEL
LIN {X 0,Y 319.519,Z 300.68,A -85,B 0,C 180,E1 -15143.323,E2 -15143.323} C_VEL
LIN {X 0,Y 319.566,Z 300.678,A -85,B 0,C 180,E1 -15146.093,E2 -15146.093} C_VEL
LIN {X 0,Y 319.526,Z 300.682,A -85,B 0,C 180,E1 -15148.939,E2 -15148.939} C_VEL
LIN {X 0,Y 319.484,Z 300.685,A -85,B 0,C 180,E1 -15151.866,E2 -15151.866} C_VEL
LIN {X 0,Y 319.542,Z 300.678,A -85,B 0,C 180,E1 -15155.546,E2 -15155.546} C_VEL
LIN {X 0,Y 319.526,Z 300.681,A -85,B 0,C 180,E1 -15159.673,E2 -15159.673} C_VEL
LIN {X 0,Y 319.489,Z 300.69,A -85,B 0,C 180,E1 -15163.464,E2 -15163.464} C_VEL
LIN {X 0,Y 319.525,Z 300.681,A -85,B 0,C 180,E1 -15167.02,E2 -15167.02} C_VEL
LIN {X 0,Y 319.52,Z 300.681,A -85,B 0,C 180,E1 -15170.375,E2 -15170.375} C_VEL
LIN {X 0,Y 319.554,Z 300.678,A -85,B 0,C 180,E1 -15174.462,E2 -15174.462} C_VEL
LIN {X 0,Y 319.575,Z 300.774,A -85,B 0,C 180,E1 -15177.685,E2 -15177.685} C_VEL
LIN {X 0,Y 322.473,Z 313.781,A -85,B 0,C 180,E1 -15180.928,E2 -15180.928} C_VEL
LIN {X 0,Y 324.868,Z 325.273,A -85,B 0,C 180,E1 -15183.679,E2 -15183.679} C_VEL
LIN {X 0,Y 324.893,Z 328.364,A -85,B 0,C 180,E1 -15184.371,E2 -15184.371} C_VEL
LIN {X 0,Y 322.931,Z 344.071,A -85,B 0,C 180,E1 -15187.745,E2 -15187.745} C_VEL
LIN {X 0,Y 325.734,Z 371.784,A -85,B 0,C 180,E1 -15188.657,E2 -15188.657} C_VEL
LIN {X 0,Y 325.729,Z 380.738,A -85,B 0,C 180,E1 -15188.905,E2 -15188.905} C_VEL
LIN {X 0,Y 324.181,Z 447.3,A -85,B 0,C 180,E1 -15190.658,E2 -15190.658} C_VEL
LIN {X 0,Y 323.781,Z 456.903,A -85,B 0,C 180,E1 -15191.044,E2 -15191.044} C_VEL
LIN {X 0,Y 323.234,Z 466.075,A -85,B 0,C 180,E1 -15191.545,E2 -15191.545} C_VEL
LIN {X 0,Y 322.542,Z 475.892,A -85,B 0,C 180,E1 -15192.243,E2 -15192.243} C_VEL
LIN {X 0,Y 321.729,Z 486.208,A -85,B 0,C 180,E1 -15193.18,E2 -15193.18} C_VEL
LIN {X 0,Y 321.066,Z 494.7,A -85,B 0,C 180,E1 -15194.125,E2 -15194.125} C_VEL
LIN {X 0,Y 320.316,Z 502.973,A -85,B 0,C 180,E1 -15195.227,E2 -15195.227} C_VEL
LIN {X 0,Y 319.752,Z 510.058,A -85,B 0,C 180,E1 -15196.337,E2 -15196.337} C_VEL
LIN {X 0,Y 319.104,Z 518.405,A -85,B 0,C 180,E1 -15197.927,E2 -15197.927} C_VEL
LIN {X 0,Y 318.586,Z 525.285,A -85,B 0,C 180,E1 -15199.518,E2 -15199.518} C_VEL
LIN {X 0,Y 318.273,Z 530.97,A -85,B 0,C 180,E1 -15201.112,E2 -15201.112} C_VEL
LIN {X 0,Y 318.133,Z 534.842,A -85,B 0,C 180,E1 -15202.386,E2 -15202.386} C_VEL
LIN {X 0,Y 318.026,Z 538.672,A -85,B 0,C 180,E1 -15203.952,E2 -15203.952} C_VEL
LIN {X 0,Y 317.965,Z 542.758,A -85,B 0,C 180,E1 -15206.201,E2 -15206.201} C_VEL
LIN {X 0,Y 317.977,Z 544.377,A -85,B 0,C 180,E1 -15207.469,E2 -15207.469} C_VEL
LIN {X 0,Y 318.12,Z 545.507,A -85,B 0,C 180,E1 -15208.737,E2 -15208.737} C_VEL
LIN {X 0,Y 318.146,Z 546.286,A -85,B 0,C 180,E1 -15210.003,E2 -15210.003} C_VEL
LIN {X 0,Y 317.974,Z 546.524,A -85,B 0,C 180,E1 -15211.269,E2 -15211.269} C_VEL
LIN {X 0,Y 317.864,Z 545.766,A -85,B 0,C 180,E1 -15213.805,E2 -15213.805} C_VEL
LIN {X 0,Y 317.855,Z 543.979,A -85,B 0,C 180,E1 -15215.75,E2 -15215.75} C_VEL
LIN {X 0,Y 318.029,Z 541.296,A -85,B 0,C 180,E1 -15217.621,E2 -15217.621} C_VEL
LIN {X 0,Y 318.412,Z 537.489,A -85,B 0,C 180,E1 -15219.53,E2 -15219.53} C_VEL
LIN {X 0,Y 319.036,Z 532.511,A -85,B 0,C 180,E1 -15221.437,E2 -15221.437} C_VEL
LIN {X 0,Y 320.124,Z 526.209,A -85,B 0,C 180,E1 -15223.329,E2 -15223.329} C_VEL
LIN {X 0,Y 321.119,Z 519.802,A -85,B 0,C 180,E1 -15224.903,E2 -15224.903} C_VEL
LIN {X 0,Y 322.213,Z 512.906,A -85,B 0,C 180,E1 -15226.321,E2 -15226.321} C_VEL
LIN {X 0,Y 323.626,Z 504.826,A -85,B 0,C 180,E1 -15227.701,E2 -15227.701} C_VEL
LIN {X 0,Y 325.035,Z 496.175,A -85,B 0,C 180,E1 -15228.926,E2 -15228.926} C_VEL
LIN {X 0,Y 326.449,Z 487.083,A -85,B 0,C 180,E1 -15229.985,E2 -15229.985} C_VEL
LIN {X 0,Y 327.79,Z 477.621,A -85,B 0,C 180,E1 -15230.883,E2 -15230.883} C_VEL
LIN {X 0,Y 328.914,Z 467.882,A -85,B 0,C 180,E1 -15231.629,E2 -15231.629} C_VEL
LIN {X 0,Y 329.89,Z 457.939,A -85,B 0,C 180,E1 -15232.219,E2 -15232.219} C_VEL
LIN {X 0,Y 330.719,Z 447.889,A -85,B 0,C 180,E1 -15232.654,E2 -15232.654} C_VEL
LIN {X 0,Y 331.951,Z 419.382,A -85,B 0,C 180,E1 -15233.472,E2 -15233.472} C_VEL
LIN {X 0,Y 333.836,Z 375.236,A -85,B 0,C 180,E1 -15234.704,E2 -15234.704} C_VEL
LIN {X 0,Y 331.685,Z 358.561,A -85,B 0,C 180,E1 -15235.514,E2 -15235.514} C_VEL
LIN {X 0,Y 328.668,Z 342.859,A -85,B 0,C 180,E1 -15236.441,E2 -15236.441} C_VEL
LIN {X 0,Y 329.581,Z 336.979,A -85,B 0,C 180,E1 -15237.632,E2 -15237.632} C_VEL
LIN {X 0,Y 328.675,Z 330.776,A -85,B 0,C 180,E1 -15239.158,E2 -15239.158} C_VEL
LIN {X 0,Y 326.444,Z 321.408,A -85,B 0,C 180,E1 -15241.716,E2 -15241.716} C_VEL
LIN {X 0,Y 323.817,Z 312.44,A -85,B 0,C 180,E1 -15244.439,E2 -15244.439} C_VEL
LIN {X 0,Y 320.854,Z 304.359,A -85,B 0,C 180,E1 -15247.259,E2 -15247.259} C_VEL
LIN {X 0,Y 319.549,Z 300.685,A -85,B 0,C 180,E1 -15248.713,E2 -15248.713} C_VEL
LIN {X 0,Y 319.545,Z 300.684,A -85,B 0,C 180,E1 -15252.983,E2 -15252.983} C_VEL
LIN {X 0,Y 319.545,Z 300.683,A -85,B 0,C 180,E1 -15257.016,E2 -15257.016} C_VEL
LIN {X 0,Y 319.572,Z 300.674,A -85,B 0,C 180,E1 -15260.375,E2 -15260.375} C_VEL
LIN {X 0,Y 319.545,Z 300.678,A -85,B 0,C 180,E1 -15263.571,E2 -15263.571} C_VEL
LIN {X 0,Y 319.564,Z 300.668,A -85,B 0,C 180,E1 -15266.686,E2 -15266.686} C_VEL
LIN {X 0,Y 319.576,Z 300.666,A -85,B 0,C 180,E1 -15269.616,E2 -15269.616} C_VEL
LIN {X 0,Y 319.592,Z 300.669,A -85,B 0,C 180,E1 -15272.497,E2 -15272.497} C_VEL
LIN {X 0,Y 319.595,Z 300.675,A -85,B 0,C 180,E1 -15275.304,E2 -15275.304} C_VEL
LIN {X 0,Y 319.612,Z 300.674,A -85,B 0,C 180,E1 -15279.402,E2 -15279.402} C_VEL
LIN {X 0,Y 319.639,Z 300.669,A -85,B 0,C 180,E1 -15282.073,E2 -15282.073} C_VEL
LIN {X 0,Y 319.704,Z 300.673,A -85,B 0,C 180,E1 -15285.686,E2 -15285.686} C_VEL
LIN {X 0,Y 323.629,Z 311.299,A -85,B 0,C 180,E1 -15289.391,E2 -15289.391} C_VEL
LIN {X 0,Y 326.719,Z 320.865,A -85,B 0,C 180,E1 -15292.244,E2 -15292.244} C_VEL
LIN {X 0,Y 328.571,Z 329.476,A -85,B 0,C 180,E1 -15294.477,E2 -15294.477} C_VEL
LIN {X 0,Y 327.537,Z 338.721,A -85,B 0,C 180,E1 -15296.352,E2 -15296.352} C_VEL
LIN {X 0,Y 331.128,Z 355.858,A -85,B 0,C 180,E1 -15297.493,E2 -15297.493} C_VEL
LIN {X 0,Y 333.431,Z 370.886,A -85,B 0,C 180,E1 -15298.34,E2 -15298.34} C_VEL
LIN {X 0,Y 330.458,Z 427.668,A -85,B 0,C 180,E1 -15300.212,E2 -15300.212} C_VEL
LIN {X 0,Y 329.614,Z 438.958,A -85,B 0,C 180,E1 -15300.764,E2 -15300.764} C_VEL
LIN {X 0,Y 328.565,Z 450.067,A -85,B 0,C 180,E1 -15301.533,E2 -15301.533} C_VEL
LIN {X 0,Y 327.419,Z 460.128,A -85,B 0,C 180,E1 -15302.461,E2 -15302.461} C_VEL
LIN {X 0,Y 326.161,Z 469.545,A -85,B 0,C 180,E1 -15303.552,E2 -15303.552} C_VEL
LIN {X 0,Y 324.838,Z 478.138,A -85,B 0,C 180,E1 -15304.781,E2 -15304.781} C_VEL
LIN {X 0,Y 323.453,Z 486.349,A -85,B 0,C 180,E1 -15306.238,E2 -15306.238} C_VEL
LIN {X 0,Y 322.147,Z 493.406,A -85,B 0,C 180,E1 -15307.837,E2 -15307.837} C_VEL
LIN {X 0,Y 321.177,Z 498.547,A -85,B 0,C 180,E1 -15309.279,E2 -15309.279} C_VEL
LIN {X 0,Y 320.331,Z 502.791,A -85,B 0,C 180,E1 -15310.749,E2 -15310.749} C_VEL
LIN {X 0,Y 319.68,Z 505.845,A -85,B 0,C 180,E1 -15312.056,E2 -15312.056} C_VEL
LIN {X 0,Y 318.963,Z 509.096,A -85,B 0,C 180,E1 -15314.027,E2 -15314.027} C_VEL
LIN {X 0,Y 318.562,Z 510.605,A -85,B 0,C 180,E1 -15315.352,E2 -15315.352} C_VEL
LIN {X 0,Y 318.233,Z 511.526,A -85,B 0,C 180,E1 -15316.685,E2 -15316.685} C_VEL
LIN {X 0,Y 318.018,Z 511.815,A -85,B 0,C 180,E1 -15318.154,E2 -15318.154} C_VEL
LIN {X 0,Y 317.906,Z 511.503,A -85,B 0,C 180,E1 -15319.367,E2 -15319.367} C_VEL
LIN {X 0,Y 317.885,Z 509.626,A -85,B 0,C 180,E1 -15321.796,E2 -15321.796} C_VEL
LIN {X 0,Y 318.037,Z 507.176,A -85,B 0,C 180,E1 -15323.439,E2 -15323.439} C_VEL
LIN {X 0,Y 318.257,Z 503.616,A -85,B 0,C 180,E1 -15325.13,E2 -15325.13} C_VEL
LIN {X 0,Y 318.582,Z 498.685,A -85,B 0,C 180,E1 -15326.888,E2 -15326.888} C_VEL
LIN {X 0,Y 318.988,Z 493.014,A -85,B 0,C 180,E1 -15328.479,E2 -15328.479} C_VEL
LIN {X 0,Y 319.494,Z 486.153,A -85,B 0,C 180,E1 -15330.03,E2 -15330.03} C_VEL
LIN {X 0,Y 320.162,Z 477.708,A -85,B 0,C 180,E1 -15331.572,E2 -15331.572} C_VEL
LIN {X 0,Y 320.932,Z 467.564,A -85,B 0,C 180,E1 -15333.007,E2 -15333.007} C_VEL
LIN {X 0,Y 321.553,Z 458.622,A -85,B 0,C 180,E1 -15334.026,E2 -15334.026} C_VEL
LIN {X 0,Y 322.17,Z 448.674,A -85,B 0,C 180,E1 -15334.935,E2 -15334.935} C_VEL
LIN {X 0,Y 322.82,Z 435.736,A -85,B 0,C 180,E1 -15335.81,E2 -15335.81} C_VEL
LIN {X 0,Y 323.186,Z 425.052,A -85,B 0,C 180,E1 -15336.302,E2 -15336.302} C_VEL
LIN {X 0,Y 324.683,Z 366.754,A -85,B 0,C 180,E1 -15338.035,E2 -15338.035} C_VEL
LIN {X 0,Y 321.347,Z 339.882,A -85,B 0,C 180,E1 -15339.008,E2 -15339.008} C_VEL
LIN {X 0,Y 322.76,Z 323.041,A -85,B 0,C 180,E1 -15343.308,E2 -15343.308} C_VEL
LIN {X 0,Y 323.013,Z 318.267,A -85,B 0,C 180,E1 -15344.558,E2 -15344.558} C_VEL
LIN {X 0,Y 320.794,Z 306.66,A -85,B 0,C 180,E1 -15347.847,E2 -15347.847} C_VEL
LIN {X 0,Y 319.56,Z 300.681,A -85,B 0,C 180,E1 -15349.656,E2 -15349.656} C_VEL
LIN {X 0,Y 319.553,Z 300.682,A -85,B 0,C 180,E1 -15353.573,E2 -15353.573} C_VEL
LIN {X 0,Y 319.578,Z 300.673,A -85,B 0,C 180,E1 -15356.688,E2 -15356.688} C_VEL
LIN {X 0,Y 319.553,Z 300.679,A -85,B 0,C 180,E1 -15359.613,E2 -15359.613} C_VEL
LIN {X 0,Y 319.535,Z 300.681,A -85,B 0,C 180,E1 -15362.491,E2 -15362.491} C_VEL
LIN {X 0,Y 319.527,Z 300.679,A -85,B 0,C 180,E1 -15365.297,E2 -15365.297} C_VEL
LIN {X 0,Y 319.567,Z 300.677,A -85,B 0,C 180,E1 -15368.045,E2 -15368.045} C_VEL
LIN {X 0,Y 319.618,Z 300.669,A -85,B 0,C 180,E1 -15372.07,E2 -15372.07} C_VEL
LIN {X 0,Y 319.736,Z 300.653,A -85,B 0,C 180,E1 -15376.007,E2 -15376.007} C_VEL
LIN {X 0,Y 319.74,Z 300.653,A -85,B 0,C 180,E1 -15379.871,E2 -15379.871} C_VEL
LIN {X 0,Y 319.902,Z 300.636,A -85,B 0,C 180,E1 -15383.692,E2 -15383.692} C_VEL
LIN {X 0,Y 319.951,Z 300.632,A -85,B 0,C 180,E1 -15387.48,E2 -15387.48} C_VEL
LIN {X 0,Y 320,Z 300.622,A -85,B 0,C 180,E1 -15391.256,E2 -15391.256} C_VEL
LIN {X 0,Y 319.691,Z 300.663,A -85,B 0,C 180,E1 -15393.779,E2 -15393.779} C_VEL
LIN {X 0,Y 319.899,Z 300.637,A -85,B 0,C 180,E1 -15396.303,E2 -15396.303} C_VEL
LIN {X 0,Y 319.735,Z 300.658,A -85,B 0,C 180,E1 -15400.124,E2 -15400.124} C_VEL
LIN {X 0,Y 319.731,Z 300.655,A -85,B 0,C 180,E1 -15403.988,E2 -15403.988} C_VEL
LIN {X 0,Y 319.61,Z 300.669,A -85,B 0,C 180,E1 -15407.925,E2 -15407.925} C_VEL
LIN {X 0,Y 319.559,Z 300.675,A -85,B 0,C 180,E1 -15411.95,E2 -15411.95} C_VEL
